LIN {X 0,Y 305.543,Z 612.418,A -85,B 0,C 180,E1 -15866.228,E2 -15866.228} C_VEL
LIN {X 0,Y 305.492,Z 612.423,A -85,B 0,C 180,E1 -15869.051,E2 -15869.051} C_VEL
LIN {X 0,Y 305.444,Z 612.427,A -85,B 0,C 180,E1 -15871.953,E2 -15871.953} C_VEL
LIN {X 0,Y 305.459,Z 612.428,A -85,B 0,C 180,E1 -15875.114,E2 -15875.114} C_VEL
LIN {X 0,Y 305.479,Z 612.428,A -85,B 0,C 180,E1 -15878.537,E2 -15878.537} C_VEL
LIN {X 0,Y 305.49,Z 612.432,A -85,B 0,C 180,E1 -15882.594,E2 -15882.594} C_VEL
LIN {X 0,Y 305.48,Z 612.432,A -85,B 0,C 180,E1 -15886.356,E2 -15886.356} C_VEL
LIN {X 0,Y 305.465,Z 612.434,A -85,B 0,C 180,E1 -15889.895,E2 -15889.895} C_VEL
LIN {X 0,Y 305.512,Z 612.46,A -85,B 0,C 180,E1 -15892.958,E2 -15892.958} C_VEL
LIN {X 0,Y 307.907,Z 621.669,A -85,B 0,C 180,E1 -15896.446,E2 -15896.446} C_VEL
LIN {X 0,Y 310.34,Z 632.372,A -85,B 0,C 180,E1 -15900.119,E2 -15900.119} C_VEL
LIN {X 0,Y 311.626,Z 639.236,A -85,B 0,C 180,E1 -15902.28,E2 -15902.28} C_VEL
LIN {X 0,Y 313.295,Z 644.798,A -85,B 0,C 180,E1 -15902.654,E2 -15902.654} C_VEL
LIN {X 0,Y 317.551,Z 667.18,A -85,B 0,C 180,E1 -15903.81,E2 -15903.81} C_VEL
LIN {X 0,Y 319.912,Z 685.577,A -85,B 0,C 180,E1 -15904.607,E2 -15904.607} C_VEL
LIN {X 0,Y 317.704,Z 749.055,A -85,B 0,C 180,E1 -15906.253,E2 -15906.253} C_VEL
LIN {X 0,Y 316.565,Z 763.423,A -85,B 0,C 180,E1 -15906.879,E2 -15906.879} C_VEL
LIN {X 0,Y 315.132,Z 776.341,A -85,B 0,C 180,E1 -15907.721,E2 -15907.721} C_VEL
LIN {X 0,Y 313.453,Z 788.638,A -85,B 0,C 180,E1 -15908.806,E2 -15908.806} C_VEL
LIN {X 0,Y 311.748,Z 799.729,A -85,B 0,C 180,E1 -15910.064,E2 -15910.064} C_VEL
LIN {X 0,Y 310.042,Z 809.772,A -85,B 0,C 180,E1 -15911.498,E2 -15911.498} C_VEL
LIN {X 0,Y 308.518,Z 818.8,A -85,B 0,C 180,E1 -15913.09,E2 -15913.09} C_VEL
LIN {X 0,Y 307.022,Z 827.902,A -85,B 0,C 180,E1 -15915.077,E2 -15915.077} C_VEL
LIN {X 0,Y 305.66,Z 835.139,A -85,B 0,C 180,E1 -15917.046,E2 -15917.046} C_VEL
LIN {X 0,Y 304.621,Z 841.793,A -85,B 0,C 180,E1 -15919.364,E2 -15919.364} C_VEL
LIN {X 0,Y 304.064,Z 846.209,A -85,B 0,C 180,E1 -15921.359,E2 -15921.359} C_VEL
LIN {X 0,Y 303.757,Z 849.545,A -85,B 0,C 180,E1 -15923.357,E2 -15923.357} C_VEL
LIN {X 0,Y 303.688,Z 851.227,A -85,B 0,C 180,E1 -15924.689,E2 -15924.689} C_VEL
LIN {X 0,Y 303.681,Z 852.481,A -85,B 0,C 180,E1 -15926.019,E2 -15926.019} C_VEL
LIN {X 0,Y 303.674,Z 853.284,A -85,B 0,C 180,E1 -15927.347,E2 -15927.347} C_VEL
LIN {X 0,Y 303.694,Z 853.688,A -85,B 0,C 180,E1 -15928.674,E2 -15928.674} C_VEL
LIN {X 0,Y 303.794,Z 853.697,A -85,B 0,C 180,E1 -15930,E2 -15930} C_VEL
LIN {X 0,Y 303.722,Z 853.275,A -85,B 0,C 180,E1 -15931.326,E2 -15931.326} C_VEL
LIN {X 0,Y 303.685,Z 852.404,A -85,B 0,C 180,E1 -15932.653,E2 -15932.653} C_VEL
LIN {X 0,Y 303.703,Z 851.122,A -85,B 0,C 180,E1 -15933.981,E2 -15933.981} C_VEL
LIN {X 0,Y 303.732,Z 848.735,A -85,B 0,C 180,E1 -15935.745,E2 -15935.745} C_VEL
LIN {X 0,Y 303.946,Z 844.524,A -85,B 0,C 180,E1 -15937.974,E2 -15937.974} C_VEL
LIN {X 0,Y 304.356,Z 839.52,A -85,B 0,C 180,E1 -15939.973,E2 -15939.973} C_VEL
LIN {X 0,Y 304.988,Z 833.193,A -85,B 0,C 180,E1 -15941.969,E2 -15941.969} C_VEL
LIN {X 0,Y 306.069,Z 825.275,A -85,B 0,C 180,E1 -15943.951,E2 -15943.951} C_VEL
LIN {X 0,Y 307.063,Z 817.151,A -85,B 0,C 180,E1 -15945.6,E2 -15945.6} C_VEL
LIN {X 0,Y 308.266,Z 807.236,A -85,B 0,C 180,E1 -15947.24,E2 -15947.24} C_VEL
LIN {X 0,Y 309.704,Z 796.205,A -85,B 0,C 180,E1 -15948.695,E2 -15948.695} C_VEL
LIN {X 0,Y 311.143,Z 783.651,A -85,B 0,C 180,E1 -15949.976,E2 -15949.976} C_VEL
LIN {X 0,Y 312.364,Z 771.376,A -85,B 0,C 180,E1 -15950.926,E2 -15950.926} C_VEL
LIN {X 0,Y 313.352,Z 758.55,A -85,B 0,C 180,E1 -15951.633,E2 -15951.633} C_VEL
LIN {X 0,Y 313.919,Z 745.321,A -85,B 0,C 180,E1 -15952.11,E2 -15952.11} C_VEL
LIN {X 0,Y 315.418,Z 683.907,A -85,B 0,C 180,E1 -15953.644,E2 -15953.644} C_VEL
LIN {X 0,Y 309.576,Z 641.497,A -85,B 0,C 180,E1 -15955.219,E2 -15955.219} C_VEL
LIN {X 0,Y 310.286,Z 636.303,A -85,B 0,C 180,E1 -15956.572,E2 -15956.572} C_VEL
LIN {X 0,Y 309.106,Z 629.471,A -85,B 0,C 180,E1 -15958.519,E2 -15958.519} C_VEL
LIN {X 0,Y 306.453,Z 617.001,A -85,B 0,C 180,E1 -15962.22,E2 -15962.22} C_VEL
LIN {X 0,Y 305.476,Z 612.433,A -85,B 0,C 180,E1 -15963.654,E2 -15963.654} C_VEL
LIN {X 0,Y 305.497,Z 612.431,A -85,B 0,C 180,E1 -15966.735,E2 -15966.735} C_VEL
LIN {X 0,Y 305.463,Z 612.438,A -85,B 0,C 180,E1 -15970.601,E2 -15970.601} C_VEL
LIN {X 0,Y 305.48,Z 612.431,A -85,B 0,C 180,E1 -15973.644,E2 -15973.644} C_VEL
LIN {X 0,Y 305.49,Z 612.429,A -85,B 0,C 180,E1 -15977.406,E2 -15977.406} C_VEL
LIN {X 0,Y 305.506,Z 612.427,A -85,B 0,C 180,E1 -15981.601,E2 -15981.601} C_VEL
LIN {X 0,Y 305.46,Z 612.438,A -85,B 0,C 180,E1 -15984.886,E2 -15984.886} C_VEL
LIN {X 0,Y 305.452,Z 612.435,A -85,B 0,C 180,E1 -15988.353,E2 -15988.353} C_VEL
LIN {X 0,Y 305.517,Z 612.429,A -85,B 0,C 180,E1 -15991.113,E2 -15991.113} C_VEL
LIN {X 0,Y 305.567,Z 612.418,A -85,B 0,C 180,E1 -15994.087,E2 -15994.087} C_VEL
LIN {X 0,Y 305.475,Z 612.431,A -85,B 0,C 180,E1 -15998.4,E2 -15998.4} C_VEL
LIN {X 0,Y 305.574,Z 612.422,A -85,B 0,C 180,E1 -16001.216,E2 -16001.216} C_VEL
LIN {X 0,Y 305.643,Z 612.414,A -85,B 0,C 180,E1 -16005.348,E2 -16005.348} C_VEL
LIN {X 0,Y 305.631,Z 612.413,A -85,B 0,C 180,E1 -16009.399,E2 -16009.399} C_VEL
LIN {X 0,Y 305.802,Z 612.389,A -85,B 0,C 180,E1 -16012.073,E2 -16012.073} C_VEL
LIN {X 0,Y 305.682,Z 612.405,A -85,B 0,C 180,E1 -16014.723,E2 -16014.723} C_VEL
LIN {X 0,Y 305.951,Z 612.371,A -85,B 0,C 180,E1 -16018.683,E2 -16018.683} C_VEL
LIN {X 0,Y 305.951,Z 612.373,A -85,B 0,C 180,E1 -16021.316,E2 -16021.316} C_VEL
LIN {X 0,Y 305.841,Z 612.385,A -85,B 0,C 180,E1 -16026.597,E2 -16026.597} C_VEL
LIN {X 0,Y 305.728,Z 612.401,A -85,B 0,C 180,E1 -16029.259,E2 -16029.259} C_VEL
LIN {X 0,Y 305.58,Z 612.416,A -85,B 0,C 180,E1 -16033.296,E2 -16033.296} C_VEL
LIN {X 0,Y 305.586,Z 612.419,A -85,B 0,C 180,E1 -16036.02,E2 -16036.02} C_VEL
LIN {X 0,Y 305.569,Z 612.421,A -85,B 0,C 180,E1 -16039.444,E2 -16039.444} C_VEL
LIN {X 0,Y 305.482,Z 612.428,A -85,B 0,C 180,E1 -16043.041,E2 -16043.041} C_VEL
LIN {X 0,Y 305.54,Z 612.423,A -85,B 0,C 180,E1 -16046.227,E2 -16046.227} C_VEL
LIN {X 0,Y 305.488,Z 612.428,A -85,B 0,C 180,E1 -16049.05,E2 -16049.05} C_VEL
LIN {X 0,Y 305.441,Z 612.439,A -85,B 0,C 180,E1 -16051.952,E2 -16051.952} C_VEL
LIN {X 0,Y 305.455,Z 612.432,A -85,B 0,C 180,E1 -16055.113,E2 -16055.113} C_VEL
LIN {X 0,Y 305.486,Z 612.429,A -85,B 0,C 180,E1 -16058.539,E2 -16058.539} C_VEL
LIN {X 0,Y 305.504,Z 612.429,A -85,B 0,C 180,E1 -16062.597,E2 -16062.597} C_VEL
LIN {X 0,Y 305.481,Z 612.434,A -85,B 0,C 180,E1 -16066.356,E2 -16066.356} C_VEL
LIN {X 0,Y 305.459,Z 612.431,A -85,B 0,C 180,E1 -16069.894,E2 -16069.894} C_VEL
LIN {X 0,Y 305.494,Z 612.428,A -85,B 0,C 180,E1 -16073.627,E2 -16073.627} C_VEL
LIN {X 0,Y 305.46,Z 612.438,A -85,B 0,C 180,E1 -16076.484,E2 -16076.484} C_VEL
LIN {X 0,Y 305.452,Z 612.431,A -85,B 0,C 180,E1 -16079.591,E2 -16079.591} C_VEL
LIN {X 0,Y 305.51,Z 612.432,A -85,B 0,C 180,E1 -16082.608,E2 -16082.608} C_VEL
LIN {X 0,Y 305.503,Z 612.427,A -85,B 0,C 180,E1 -16085.539,E2 -16085.539} C_VEL
LIN {X 0,Y 305.516,Z 612.425,A -85,B 0,C 180,E1 -16089.815,E2 -16089.815} C_VEL
LIN {X 0,Y 305.571,Z 612.423,A -85,B 0,C 180,E1 -16092.603,E2 -16092.603} C_VEL
LIN {X 0,Y 305.645,Z 612.41,A -85,B 0,C 180,E1 -16095.349,E2 -16095.349} C_VEL
LIN {X 0,Y 305.635,Z 612.411,A -85,B 0,C 180,E1 -16099.4,E2 -16099.4} C_VEL
LIN {X 0,Y 305.805,Z 612.389,A -85,B 0,C 180,E1 -16102.074,E2 -16102.074} C_VEL
LIN {X 0,Y 305.685,Z 612.407,A -85,B 0,C 180,E1 -16104.724,E2 -16104.724} C_VEL
LIN {X 0,Y 305.955,Z 612.373,A -85,B 0,C 180,E1 -16108.684,E2 -16108.684} C_VEL
LIN {X 0,Y 305.955,Z 612.374,A -85,B 0,C 180,E1 -16111.316,E2 -16111.316} C_VEL
LIN {X 0,Y 305.684,Z 612.409,A -85,B 0,C 180,E1 -16115.276,E2 -16115.276} C_VEL
LIN {X 0,Y 305.793,Z 612.392,A -85,B 0,C 180,E1 -16117.926,E2 -16117.926} C_VEL
LIN {X 0,Y 305.6,Z 612.416,A -85,B 0,C 180,E1 -16121.945,E2 -16121.945} C_VEL
LIN {X 0,Y 305.634,Z 612.415,A -85,B 0,C 180,E1 -16125.035,E2 -16125.035} C_VEL
LIN {X 0,Y 305.633,Z 612.47,A -85,B 0,C 180,E1 -16129.167,E2 -16129.167} C_VEL
LIN {X 0,Y 305.85,Z 613.833,A -85,B 0,C 180,E1 -16129.639,E2 -16129.639} C_VEL
LIN {X 0,Y 316.129,Z 642.397,A -85,B 0,C 180,E1 -16131.156,E2 -16131.156} C_VEL
LIN {X 0,Y 315.453,Z 671.633,A -85,B 0,C 180,E1 -16131.889,E2 -16131.889} C_VEL
LIN {X 0,Y 313.978,Z 721.477,A -85,B 0,C 180,E1 -16133.152,E2 -16133.152} C_VEL
LIN {X 0,Y 313.316,Z 735.297,A -85,B 0,C 180,E1 -16133.778,E2 -16133.778} C_VEL
LIN {X 0,Y 312.468,Z 747.528,A -85,B 0,C 180,E1 -16134.588,E2 -16134.588} C_VEL
LIN {X 0,Y 311.433,Z 758.765,A -85,B 0,C 180,E1 -16135.576,E2 -16135.576} C_VEL
LIN {X 0,Y 310.359,Z 769.3,A -85,B 0,C 180,E1 -16136.751,E2 -16136.751} C_VEL
LIN {X 0,Y 309.152,Z 778.865,A -85,B 0,C 180,E1 -16138.06,E2 -16138.06} C_VEL
LIN {X 0,Y 308.068,Z 788.02,A -85,B 0,C 180,E1 -16139.597,E2 -16139.597} C_VEL
LIN {X 0,Y 306.895,Z 796.747,A -85,B 0,C 180,E1 -16141.397,E2 -16141.397} C_VEL
LIN {X 0,Y 305.795,Z 804.771,A -85,B 0,C 180,E1 -16143.475,E2 -16143.475} C_VEL
LIN {X 0,Y 304.953,Z 811.468,A -85,B 0,C 180,E1 -16145.676,E2 -16145.676} C_VEL
LIN {X 0,Y 304.418,Z 815.911,A -85,B 0,C 180,E1 -16147.554,E2 -16147.554} C_VEL
LIN {X 0,Y 304.021,Z 819.316,A -85,B 0,C 180,E1 -16149.417,E2 -16149.417} C_VEL
LIN {X 0,Y 303.747,Z 821.79,A -85,B 0,C 180,E1 -16151.255,E2 -16151.255} C_VEL
LIN {X 0,Y 303.507,Z 823.992,A -85,B 0,C 180,E1 -16154,E2 -16154} C_VEL
LIN {X 0,Y 303.51,Z 824.497,A -85,B 0,C 180,E1 -16156,E2 -16156} C_VEL
LIN {X 0,Y 303.647,Z 824.132,A -85,B 0,C 180,E1 -16157.84,E2 -16157.84} C_VEL
LIN {X 0,Y 303.992,Z 822.94,A -85,B 0,C 180,E1 -16159.721,E2 -16159.721} C_VEL
LIN {X 0,Y 304.443,Z 820.788,A -85,B 0,C 180,E1 -16161.708,E2 -16161.708} C_VEL
LIN {X 0,Y 305.069,Z 817.577,A -85,B 0,C 180,E1 -16163.735,E2 -16163.735} C_VEL
LIN {X 0,Y 306.122,Z 812.196,A -85,B 0,C 180,E1 -16166.19,E2 -16166.19} C_VEL
LIN {X 0,Y 307.281,Z 806.133,A -85,B 0,C 180,E1 -16168.262,E2 -16168.262} C_VEL
LIN {X 0,Y 308.82,Z 798.31,A -85,B 0,C 180,E1 -16170.361,E2 -16170.361} C_VEL
LIN {X 0,Y 310.445,Z 789.859,A -85,B 0,C 180,E1 -16172.164,E2 -16172.164} C_VEL
LIN {X 0,Y 311.242,Z 785.111,A -85,B 0,C 180,E1 -16173.023,E2 -16173.023} C_VEL
LIN {X 0,Y 311.3,Z 780.871,A -85,B 0,C 180,E1 -16173.773,E2 -16173.773} C_VEL
LIN {X 0,Y 309.142,Z 770.889,A -85,B 0,C 180,E1 -16175.515,E2 -16175.515} C_VEL
LIN {X 0,Y 308.347,Z 764.725,A -85,B 0,C 180,E1 -16176.411,E2 -16176.411} C_VEL
LIN {X 0,Y 308.54,Z 761.356,A -85,B 0,C 180,E1 -16176.796,E2 -16176.796} C_VEL
LIN {X 0,Y 310.052,Z 749.256,A -85,B 0,C 180,E1 -16177.895,E2 -16177.895} C_VEL
LIN {X 0,Y 311.225,Z 735.781,A -85,B 0,C 180,E1 -16178.795,E2 -16178.795} C_VEL
LIN {X 0,Y 312.046,Z 722.907,A -85,B 0,C 180,E1 -16179.377,E2 -16179.377} C_VEL
LIN {X 0,Y 314.81,Z 649.184,A -85,B 0,C 180,E1 -16181.33,E2 -16181.33} C_VEL
LIN {X 0,Y 308.378,Z 634.264,A -85,B 0,C 180,E1 -16182.569,E2 -16182.569} C_VEL
LIN {X 0,Y 301.448,Z 620.861,A -85,B 0,C 180,E1 -16183.918,E2 -16183.918} C_VEL
LIN {X 0,Y 299.513,Z 617.125,A -85,B 0,C 180,E1 -16184.346,E2 -16184.346} C_VEL
LIN {X 0,Y 298.551,Z 613.297,A -85,B 0,C 180,E1 -16186.212,E2 -16186.212} C_VEL
LIN {X 0,Y 298.753,Z 613.274,A -85,B 0,C 180,E1 -16191.115,E2 -16191.115} C_VEL
LIN {X 0,Y 298.792,Z 613.269,A -85,B 0,C 180,E1 -16193.247,E2 -16193.247} C_VEL
LIN {X 0,Y 298.85,Z 613.26,A -85,B 0,C 180,E1 -16197.305,E2 -16197.305} C_VEL
LIN {X 0,Y 299.019,Z 613.238,A -85,B 0,C 180,E1 -16200.001,E2 -16200.001} C_VEL
LIN {X 0,Y 298.842,Z 613.262,A -85,B 0,C 180,E1 -16202.697,E2 -16202.697} C_VEL
LIN {X 0,Y 298.793,Z 613.262,A -85,B 0,C 180,E1 -16206.755,E2 -16206.755} C_VEL
LIN {X 0,Y 298.675,Z 613.275,A -85,B 0,C 180,E1 -16209.481,E2 -16209.481} C_VEL
LIN {X 0,Y 298.547,Z 613.294,A -85,B 0,C 180,E1 -16213.616,E2 -16213.616} C_VEL
LIN {X 0,Y 298.543,Z 613.29,A -85,B 0,C 180,E1 -16216.41,E2 -16216.41} C_VEL
LIN {X 0,Y 298.506,Z 613.297,A -85,B 0,C 180,E1 -16219.656,E2 -16219.656} C_VEL
LIN {X 0,Y 298.453,Z 613.307,A -85,B 0,C 180,E1 -16223.599,E2 -16223.599} C_VEL
LIN {X 0,Y 298.485,Z 613.298,A -85,B 0,C 180,E1 -16226.575,E2 -16226.575} C_VEL
LIN {X 0,Y 298.418,Z 613.306,A -85,B 0,C 180,E1 -16229.642,E2 -16229.642} C_VEL
LIN {X 0,Y 298.394,Z 613.308,A -85,B 0,C 180,E1 -16232.801,E2 -16232.801} C_VEL
LIN {X 0,Y 298.462,Z 613.306,A -85,B 0,C 180,E1 -16236.814,E2 -16236.814} C_VEL
LIN {X 0,Y 298.416,Z 613.308,A -85,B 0,C 180,E1 -16241.096,E2 -16241.096} C_VEL
LIN {X 0,Y 298.416,Z 613.315,A -85,B 0,C 180,E1 -16245.048,E2 -16245.048} C_VEL
LIN {X 0,Y 298.419,Z 613.314,A -85,B 0,C 180,E1 -16248.746,E2 -16248.746} C_VEL
LIN {X 0,Y 298.467,Z 613.386,A -85,B 0,C 180,E1 -16252.091,E2 -16252.091} C_VEL
LIN {X 0,Y 301.004,Z 623.033,A -85,B 0,C 180,E1 -16255.92,E2 -16255.92} C_VEL
LIN {X 0,Y 303.174,Z 632.6,A -85,B 0,C 180,E1 -16259.338,E2 -16259.338} C_VEL
LIN {X 0,Y 304.453,Z 638.904,A -85,B 0,C 180,E1 -16261.378,E2 -16261.378} C_VEL
LIN {X 0,Y 307.133,Z 645.608,A -85,B 0,C 180,E1 -16261.934,E2 -16261.934} C_VEL
LIN {X 0,Y 310.973,Z 665.162,A -85,B 0,C 180,E1 -16263.018,E2 -16263.018} C_VEL
LIN {X 0,Y 313.303,Z 682.326,A -85,B 0,C 180,E1 -16263.804,E2 -16263.804} C_VEL
LIN {X 0,Y 313.776,Z 686.682,A -85,B 0,C 180,E1 -16263.987,E2 -16263.987} C_VEL
LIN {X 0,Y 311.45,Z 748.992,A -85,B 0,C 180,E1 -16265.642,E2 -16265.642} C_VEL
LIN {X 0,Y 310.314,Z 762.71,A -85,B 0,C 180,E1 -16266.253,E2 -16266.253} C_VEL
LIN {X 0,Y 308.881,Z 775.201,A -85,B 0,C 180,E1 -16267.068,E2 -16267.068} C_VEL
LIN {X 0,Y 307.143,Z 787.602,A -85,B 0,C 180,E1 -16268.172,E2 -16268.172} C_VEL
LIN {X 0,Y 305.355,Z 798.807,A -85,B 0,C 180,E1 -16269.453,E2 -16269.453} C_VEL
LIN {X 0,Y 303.516,Z 808.983,A -85,B 0,C 180,E1 -16270.91,E2 -16270.91} C_VEL
LIN {X 0,Y 301.801,Z 818.419,A -85,B 0,C 180,E1 -16272.598,E2 -16272.598} C_VEL
LIN {X 0,Y 300.335,Z 826.557,A -85,B 0,C 180,E1 -16274.389,E2 -16274.389} C_VEL
LIN {X 0,Y 298.948,Z 833.99,A -85,B 0,C 180,E1 -16276.403,E2 -16276.403} C_VEL
LIN {X 0,Y 297.852,Z 839.972,A -85,B 0,C 180,E1 -16278.43,E2 -16278.43} C_VEL
LIN {X 0,Y 297.198,Z 844.71,A -85,B 0,C 180,E1 -16280.472,E2 -16280.472} C_VEL
LIN {X 0,Y 296.789,Z 848.348,A -85,B 0,C 180,E1 -16282.517,E2 -16282.517} C_VEL
LIN {X 0,Y 296.603,Z 850.97,A -85,B 0,C 180,E1 -16284.561,E2 -16284.561} C_VEL
LIN {X 0,Y 296.596,Z 852.183,A -85,B 0,C 180,E1 -16285.924,E2 -16285.924} C_VEL
LIN {X 0,Y 296.597,Z 852.965,A -85,B 0,C 180,E1 -16287.284,E2 -16287.284} C_VEL
LIN {X 0,Y 296.607,Z 853.349,A -85,B 0,C 180,E1 -16288.642,E2 -16288.642} C_VEL
LIN {X 0,Y 296.702,Z 853.337,A -85,B 0,C 180,E1 -16290,E2 -16290} C_VEL
LIN {X 0,Y 296.633,Z 852.871,A -85,B 0,C 180,E1 -16291.358,E2 -16291.358} C_VEL
LIN {X 0,Y 296.608,Z 851.976,A -85,B 0,C 180,E1 -16292.716,E2 -16292.716} C_VEL
LIN {X 0,Y 296.616,Z 850.67,A -85,B 0,C 180,E1 -16294.076,E2 -16294.076} C_VEL
LIN {X 0,Y 296.631,Z 848.565,A -85,B 0,C 180,E1 -16295.672,E2 -16295.672} C_VEL
LIN {X 0,Y 296.885,Z 843.967,A -85,B 0,C 180,E1 -16298.165,E2 -16298.165} C_VEL
LIN {X 0,Y 297.341,Z 838.904,A -85,B 0,C 180,E1 -16300.211,E2 -16300.211} C_VEL
LIN {X 0,Y 298.007,Z 832.506,A -85,B 0,C 180,E1 -16302.254,E2 -16302.254} C_VEL
LIN {X 0,Y 299.085,Z 824.47,A -85,B 0,C 180,E1 -16304.284,E2 -16304.284} C_VEL
LIN {X 0,Y 300.065,Z 816.867,A -85,B 0,C 180,E1 -16305.856,E2 -16305.856} C_VEL
LIN {X 0,Y 301.422,Z 806.228,A -85,B 0,C 180,E1 -16307.644,E2 -16307.644} C_VEL
LIN {X 0,Y 302.906,Z 794.975,A -85,B 0,C 180,E1 -16309.13,E2 -16309.13} C_VEL
LIN {X 0,Y 304.245,Z 783.988,A -85,B 0,C 180,E1 -16310.273,E2 -16310.273} C_VEL
LIN {X 0,Y 305.496,Z 771.915,A -85,B 0,C 180,E1 -16311.243,E2 -16311.243} C_VEL
LIN {X 0,Y 306.506,Z 759.574,A -85,B 0,C 180,E1 -16311.964,E2 -16311.964} C_VEL
LIN {X 0,Y 307.153,Z 745.761,A -85,B 0,C 180,E1 -16312.491,E2 -16312.491} C_VEL
LIN {X 0,Y 308.682,Z 684.406,A -85,B 0,C 180,E1 -16314.064,E2 -16314.064} C_VEL
LIN {X 0,Y 302.771,Z 641.232,A -85,B 0,C 180,E1 -16315.711,E2 -16315.711} C_VEL
LIN {X 0,Y 303.276,Z 636.934,A -85,B 0,C 180,E1 -16316.864,E2 -16316.864} C_VEL
LIN {X 0,Y 301.412,Z 627.069,A -85,B 0,C 180,E1 -16319.764,E2 -16319.764} C_VEL
LIN {X 0,Y 298.431,Z 613.311,A -85,B 0,C 180,E1 -16324.058,E2 -16324.058} C_VEL
LIN {X 0,Y 298.439,Z 613.307,A -85,B 0,C 180,E1 -16327.753,E2 -16327.753} C_VEL
LIN {X 0,Y 298.419,Z 613.311,A -85,B 0,C 180,E1 -16331.254,E2 -16331.254} C_VEL
LIN {X 0,Y 298.415,Z 613.313,A -85,B 0,C 180,E1 -16335.046,E2 -16335.046} C_VEL
LIN {X 0,Y 298.416,Z 613.314,A -85,B 0,C 180,E1 -16338.904,E2 -16338.904} C_VEL
LIN {X 0,Y 298.464,Z 613.307,A -85,B 0,C 180,E1 -16343.186,E2 -16343.186} C_VEL
LIN {X 0,Y 298.394,Z 613.315,A -85,B 0,C 180,E1 -16347.199,E2 -16347.199} C_VEL
LIN {X 0,Y 298.429,Z 613.311,A -85,B 0,C 180,E1 -16350.613,E2 -16350.613} C_VEL
LIN {X 0,Y 298.48,Z 613.302,A -85,B 0,C 180,E1 -16353.473,E2 -16353.473} C_VEL
LIN {X 0,Y 298.426,Z 613.311,A -85,B 0,C 180,E1 -16356.699,E2 -16356.699} C_VEL
LIN {X 0,Y 298.52,Z 613.299,A -85,B 0,C 180,E1 -16360.755,E2 -16360.755} C_VEL
LIN {X 0,Y 298.587,Z 613.292,A -85,B 0,C 180,E1 -16364.994,E2 -16364.994} C_VEL
LIN {X 0,Y 298.587,Z 613.293,A -85,B 0,C 180,E1 -16369.146,E2 -16369.146} C_VEL
LIN {X 0,Y 298.748,Z 613.268,A -85,B 0,C 180,E1 -16371.885,E2 -16371.885} C_VEL
LIN {X 0,Y 298.653,Z 613.281,A -85,B 0,C 180,E1 -16374.598,E2 -16374.598} C_VEL
LIN {X 0,Y 298.918,Z 613.247,A -85,B 0,C 180,E1 -16378.652,E2 -16378.652} C_VEL
LIN {X 0,Y 298.918,Z 613.249,A -85,B 0,C 180,E1 -16381.347,E2 -16381.347} C_VEL
LIN {X 0,Y 298.787,Z 613.264,A -85,B 0,C 180,E1 -16386.753,E2 -16386.753} C_VEL
LIN {X 0,Y 298.673,Z 613.282,A -85,B 0,C 180,E1 -16389.48,E2 -16389.48} C_VEL
LIN {X 0,Y 298.544,Z 613.294,A -85,B 0,C 180,E1 -16393.615,E2 -16393.615} C_VEL
LIN {X 0,Y 298.541,Z 613.294,A -85,B 0,C 180,E1 -16396.408,E2 -16396.408} C_VEL
LIN {X 0,Y 298.504,Z 613.303,A -85,B 0,C 180,E1 -16399.654,E2 -16399.654} C_VEL
LIN {X 0,Y 298.45,Z 613.307,A -85,B 0,C 180,E1 -16403.598,E2 -16403.598} C_VEL
LIN {X 0,Y 298.482,Z 613.299,A -85,B 0,C 180,E1 -16406.574,E2 -16406.574} C_VEL
LIN {X 0,Y 298.414,Z 613.311,A -85,B 0,C 180,E1 -16409.641,E2 -16409.641} C_VEL
LIN {X 0,Y 298.39,Z 613.313,A -85,B 0,C 180,E1 -16412.8,E2 -16412.8} C_VEL
LIN {X 0,Y 298.463,Z 613.301,A -85,B 0,C 180,E1 -16416.814,E2 -16416.814} C_VEL
LIN {X 0,Y 298.446,Z 613.305,A -85,B 0,C 180,E1 -16421.25,E2 -16421.25} C_VEL
LIN {X 0,Y 298.411,Z 613.31,A -85,B 0,C 180,E1 -16425.047,E2 -16425.047} C_VEL
LIN {X 0,Y 298.414,Z 613.309,A -85,B 0,C 180,E1 -16428.745,E2 -16428.745} C_VEL
LIN {X 0,Y 298.433,Z 613.31,A -85,B 0,C 180,E1 -16432.246,E2 -16432.246} C_VEL
LIN {X 0,Y 298.403,Z 613.312,A -85,B 0,C 180,E1 -16435.581,E2 -16435.581} C_VEL
LIN {X 0,Y 298.386,Z 613.314,A -85,B 0,C 180,E1 -16438.791,E2 -16438.791} C_VEL
LIN {X 0,Y 298.452,Z 613.305,A -85,B 0,C 180,E1 -16441.904,E2 -16441.904} C_VEL
LIN {X 0,Y 298.479,Z 613.304,A -85,B 0,C 180,E1 -16444.924,E2 -16444.924} C_VEL
LIN {X 0,Y 298.446,Z 613.307,A -85,B 0,C 180,E1 -16449.316,E2 -16449.316} C_VEL
LIN {X 0,Y 298.534,Z 613.296,A -85,B 0,C 180,E1 -16452.18,E2 -16452.18} C_VEL
LIN {X 0,Y 298.59,Z 613.291,A -85,B 0,C 180,E1 -16454.995,E2 -16454.995} C_VEL
LIN {X 0,Y 298.59,Z 613.291,A -85,B 0,C 180,E1 -16459.147,E2 -16459.147} C_VEL
LIN {X 0,Y 298.751,Z 613.267,A -85,B 0,C 180,E1 -16461.886,E2 -16461.886} C_VEL
LIN {X 0,Y 298.655,Z 613.282,A -85,B 0,C 180,E1 -16464.599,E2 -16464.599} C_VEL
LIN {X 0,Y 298.921,Z 613.248,A -85,B 0,C 180,E1 -16468.653,E2 -16468.653} C_VEL
LIN {X 0,Y 298.921,Z 613.25,A -85,B 0,C 180,E1 -16471.347,E2 -16471.347} C_VEL
LIN {X 0,Y 298.784,Z 613.266,A -85,B 0,C 180,E1 -16476.754,E2 -16476.754} C_VEL
LIN {X 0,Y 298.632,Z 613.287,A -85,B 0,C 180,E1 -16479.482,E2 -16479.482} C_VEL
LIN {X 0,Y 298.549,Z 613.298,A -85,B 0,C 180,E1 -16483.615,E2 -16483.615} C_VEL
LIN {X 0,Y 298.546,Z 613.295,A -85,B 0,C 180,E1 -16486.408,E2 -16486.408} C_VEL
LIN {X 0,Y 298.577,Z 613.417,A -85,B 0,C 180,E1 -16488.839,E2 -16488.839} C_VEL
LIN {X 0,Y 298.714,Z 614.142,A -85,B 0,C 180,E1 -16489.097,E2 -16489.097} C_VEL
LIN {X 0,Y 309.479,Z 643.855,A -85,B 0,C 180,E1 -16490.739,E2 -16490.739} C_VEL
LIN {X 0,Y 307.27,Z 721.207,A -85,B 0,C 180,E1 -16492.73,E2 -16492.73} C_VEL
LIN {X 0,Y 306.588,Z 734.937,A -85,B 0,C 180,E1 -16493.354,E2 -16493.354} C_VEL
LIN {X 0,Y 305.698,Z 747.493,A -85,B 0,C 180,E1 -16494.189,E2 -16494.189} C_VEL
LIN {X 0,Y 304.559,Z 759.516,A -85,B 0,C 180,E1 -16495.271,E2 -16495.271} C_VEL
LIN {X 0,Y 303.43,Z 770.04,A -85,B 0,C 180,E1 -16496.478,E2 -16496.478} C_VEL
LIN {X 0,Y 302.143,Z 779.991,A -85,B 0,C 180,E1 -16497.885,E2 -16497.885} C_VEL
LIN {X 0,Y 301.104,Z 788.435,A -85,B 0,C 180,E1 -16499.35,E2 -16499.35} C_VEL
LIN {X 0,Y 299.82,Z 797.74,A -85,B 0,C 180,E1 -16501.336,E2 -16501.336} C_VEL
LIN {X 0,Y 298.847,Z 804.585,A -85,B 0,C 180,E1 -16503.145,E2 -16503.145} C_VEL
LIN {X 0,Y 298.005,Z 811.107,A -85,B 0,C 180,E1 -16505.294,E2 -16505.294} C_VEL
LIN {X 0,Y 297.429,Z 815.684,A -85,B 0,C 180,E1 -16507.209,E2 -16507.209} C_VEL
LIN {X 0,Y 297.076,Z 818.523,A -85,B 0,C 180,E1 -16508.677,E2 -16508.677} C_VEL
LIN {X 0,Y 296.71,Z 821.532,A -85,B 0,C 180,E1 -16510.716,E2 -16510.716} C_VEL
LIN {X 0,Y 296.425,Z 823.996,A -85,B 0,C 180,E1 -16513.436,E2 -16513.436} C_VEL
LIN {X 0,Y 296.381,Z 824.753,A -85,B 0,C 180,E1 -16515.346,E2 -16515.346} C_VEL
LIN {X 0,Y 296.489,Z 824.712,A -85,B 0,C 180,E1 -16517.291,E2 -16517.291} C_VEL
LIN {X 0,Y 296.814,Z 823.82,A -85,B 0,C 180,E1 -16519.26,E2 -16519.26} C_VEL
LIN {X 0,Y 297.264,Z 821.997,A -85,B 0,C 180,E1 -16521.277,E2 -16521.277} C_VEL
LIN {X 0,Y 298.04,Z 818.231,A -85,B 0,C 180,E1 -16523.878,E2 -16523.878} C_VEL
LIN {X 0,Y 298.995,Z 813.721,A -85,B 0,C 180,E1 -16526.066,E2 -16526.066} C_VEL
LIN {X 0,Y 300.229,Z 807.64,A -85,B 0,C 180,E1 -16528.314,E2 -16528.314} C_VEL
LIN {X 0,Y 301.825,Z 799.991,A -85,B 0,C 180,E1 -16530.485,E2 -16530.485} C_VEL
LIN {X 0,Y 303.604,Z 791.35,A -85,B 0,C 180,E1 -16532.422,E2 -16532.422} C_VEL
LIN {X 0,Y 305.235,Z 782.329,A -85,B 0,C 180,E1 -16534.058,E2 -16534.058} C_VEL
LIN {X 0,Y 307.102,Z 771.099,A -85,B 0,C 180,E1 -16535.675,E2 -16535.675} C_VEL
LIN {X 0,Y 308.54,Z 761.356,A -85,B 0,C 180,E1 -16536.796,E2 -16536.796} C_VEL
LIN {X 0,Y 308.675,Z 756.268,A -85,B 0,C 180,E1 -16537.352,E2 -16537.352} C_VEL
LIN {X 0,Y 307.227,Z 747.915,A -85,B 0,C 180,E1 -16538.302,E2 -16538.302} C_VEL
LIN {X 0,Y 305.534,Z 739.304,A -85,B 0,C 180,E1 -16539.165,E2 -16539.165} C_VEL
LIN {X 0,Y 305.17,Z 733.808,A -85,B 0,C 180,E1 -16539.565,E2 -16539.565} C_VEL
LIN {X 0,Y 306.01,Z 720.628,A -85,B 0,C 180,E1 -16540.108,E2 -16540.108} C_VEL
LIN {X 0,Y 308.78,Z 651.206,A -85,B 0,C 180,E1 -16541.978,E2 -16541.978} C_VEL
LIN {X 0,Y 302.791,Z 637.387,A -85,B 0,C 180,E1 -16543.178,E2 -16543.178} C_VEL
LIN {X 0,Y 296.387,Z 624.948,A -85,B 0,C 180,E1 -16544.488,E2 -16544.488} C_VEL
LIN {X 0,Y 292.396,Z 617.603,A -85,B 0,C 180,E1 -16545.383,E2 -16545.383} C_VEL
LIN {X 0,Y 291.487,Z 614.177,A -85,B 0,C 180,E1 -16547.114,E2 -16547.114} C_VEL
LIN {X 0,Y 291.702,Z 614.152,A -85,B 0,C 180,E1 -16551.689,E2 -16551.689} C_VEL
LIN {X 0,Y 291.629,Z 614.157,A -85,B 0,C 180,E1 -16554.469,E2 -16554.469} C_VEL
LIN {X 0,Y 291.888,Z 614.124,A -85,B 0,C 180,E1 -16558.621,E2 -16558.621} C_VEL
LIN {X 0,Y 291.887,Z 614.123,A -85,B 0,C 180,E1 -16561.38,E2 -16561.38} C_VEL
LIN {X 0,Y 291.741,Z 614.14,A -85,B 0,C 180,E1 -16566.919,E2 -16566.919} C_VEL
LIN {X 0,Y 291.624,Z 614.153,A -85,B 0,C 180,E1 -16569.713,E2 -16569.713} C_VEL
LIN {X 0,Y 291.517,Z 614.172,A -85,B 0,C 180,E1 -16573.951,E2 -16573.951} C_VEL
LIN {X 0,Y 291.481,Z 614.172,A -85,B 0,C 180,E1 -16576.819,E2 -16576.819} C_VEL
LIN {X 0,Y 291.446,Z 614.178,A -85,B 0,C 180,E1 -16579.876,E2 -16579.876} C_VEL
LIN {X 0,Y 291.396,Z 614.186,A -85,B 0,C 180,E1 -16584.206,E2 -16584.206} C_VEL
LIN {X 0,Y 291.419,Z 614.184,A -85,B 0,C 180,E1 -16587.273,E2 -16587.273} C_VEL
LIN {X 0,Y 291.336,Z 614.191,A -85,B 0,C 180,E1 -16590.438,E2 -16590.438} C_VEL
LIN {X 0,Y 291.342,Z 614.191,A -85,B 0,C 180,E1 -16593.699,E2 -16593.699} C_VEL
LIN {X 0,Y 291.395,Z 614.183,A -85,B 0,C 180,E1 -16597.261,E2 -16597.261} C_VEL
LIN {X 0,Y 291.374,Z 614.185,A -85,B 0,C 180,E1 -16600.636,E2 -16600.636} C_VEL
LIN {X 0,Y 291.341,Z 614.195,A -85,B 0,C 180,E1 -16604.393,E2 -16604.393} C_VEL
LIN {X 0,Y 291.356,Z 614.192,A -85,B 0,C 180,E1 -16608.399,E2 -16608.399} C_VEL
LIN {X 0,Y 291.411,Z 614.359,A -85,B 0,C 180,E1 -16611.169,E2 -16611.169} C_VEL
LIN {X 0,Y 293.577,Z 622.215,A -85,B 0,C 180,E1 -16614.483,E2 -16614.483} C_VEL
LIN {X 0,Y 295.546,Z 630.518,A -85,B 0,C 180,E1 -16617.654,E2 -16617.654} C_VEL
LIN {X 0,Y 297.187,Z 638.246,A -85,B 0,C 180,E1 -16620.376,E2 -16620.376} C_VEL
LIN {X 0,Y 301.483,Z 648.322,A -85,B 0,C 180,E1 -16621.302,E2 -16621.302} C_VEL
LIN {X 0,Y 305.073,Z 666.958,A -85,B 0,C 180,E1 -16622.366,E2 -16622.366} C_VEL
LIN {X 0,Y 307.223,Z 683.292,A -85,B 0,C 180,E1 -16623.147,E2 -16623.147} C_VEL
LIN {X 0,Y 307.616,Z 688.615,A -85,B 0,C 180,E1 -16623.361,E2 -16623.361} C_VEL
LIN {X 0,Y 305.25,Z 748.282,A -85,B 0,C 180,E1 -16624.973,E2 -16624.973} C_VEL
LIN {X 0,Y 304.13,Z 762.139,A -85,B 0,C 180,E1 -16625.603,E2 -16625.603} C_VEL
LIN {X 0,Y 302.683,Z 774.186,A -85,B 0,C 180,E1 -16626.389,E2 -16626.389} C_VEL
LIN {X 0,Y 300.841,Z 786.731,A -85,B 0,C 180,E1 -16627.51,E2 -16627.51} C_VEL
LIN {X 0,Y 298.995,Z 797.996,A -85,B 0,C 180,E1 -16628.815,E2 -16628.815} C_VEL
LIN {X 0,Y 297.011,Z 808.245,A -85,B 0,C 180,E1 -16630.295,E2 -16630.295} C_VEL
LIN {X 0,Y 295.236,Z 817.506,A -85,B 0,C 180,E1 -16631.974,E2 -16631.974} C_VEL
LIN {X 0,Y 293.462,Z 826.597,A -85,B 0,C 180,E1 -16634.014,E2 -16634.014} C_VEL
LIN {X 0,Y 292.024,Z 833.962,A -85,B 0,C 180,E1 -16636.075,E2 -16636.075} C_VEL
LIN {X 0,Y 290.871,Z 839.869,A -85,B 0,C 180,E1 -16638.149,E2 -16638.149} C_VEL
LIN {X 0,Y 290.155,Z 844.549,A -85,B 0,C 180,E1 -16640.239,E2 -16640.239} C_VEL
LIN {X 0,Y 289.717,Z 848.138,A -85,B 0,C 180,E1 -16642.333,E2 -16642.333} C_VEL
LIN {X 0,Y 289.519,Z 850.717,A -85,B 0,C 180,E1 -16644.428,E2 -16644.428} C_VEL
LIN {X 0,Y 289.494,Z 851.886,A -85,B 0,C 180,E1 -16645.824,E2 -16645.824} C_VEL
LIN {X 0,Y 289.521,Z 852.648,A -85,B 0,C 180,E1 -16647.217,E2 -16647.217} C_VEL
LIN {X 0,Y 289.522,Z 853.011,A -85,B 0,C 180,E1 -16648.609,E2 -16648.609} C_VEL
LIN {X 0,Y 289.61,Z 852.971,A -85,B 0,C 180,E1 -16650,E2 -16650} C_VEL
LIN {X 0,Y 289.547,Z 852.466,A -85,B 0,C 180,E1 -16651.391,E2 -16651.391} C_VEL
LIN {X 0,Y 289.533,Z 851.55,A -85,B 0,C 180,E1 -16652.783,E2 -16652.783} C_VEL
LIN {X 0,Y 289.532,Z 850.219,A -85,B 0,C 180,E1 -16654.176,E2 -16654.176} C_VEL
LIN {X 0,Y 289.579,Z 847.354,A -85,B 0,C 180,E1 -16656.269,E2 -16656.269} C_VEL
LIN {X 0,Y 289.842,Z 843.41,A -85,B 0,C 180,E1 -16658.365,E2 -16658.365} C_VEL
LIN {X 0,Y 290.407,Z 837.294,A -85,B 0,C 180,E1 -16660.81,E2 -16660.81} C_VEL
LIN {X 0,Y 291.242,Z 830.55,A -85,B 0,C 180,E1 -16662.897,E2 -16662.897} C_VEL
LIN {X 0,Y 292.387,Z 822.157,A -85,B 0,C 180,E1 -16664.974,E2 -16664.974} C_VEL
LIN {X 0,Y 293.472,Z 813.517,A -85,B 0,C 180,E1 -16666.7,E2 -16666.7} C_VEL
LIN {X 0,Y 294.892,Z 802.847,A -85,B 0,C 180,E1 -16668.407,E2 -16668.407} C_VEL
LIN {X 0,Y 296.345,Z 792.319,A -85,B 0,C 180,E1 -16669.751,E2 -16669.751} C_VEL
LIN {X 0,Y 297.71,Z 780.738,A -85,B 0,C 180,E1 -16670.919,E2 -16670.919} C_VEL
LIN {X 0,Y 299.017,Z 767.546,A -85,B 0,C 180,E1 -16671.908,E2 -16671.908} C_VEL
LIN {X 0,Y 300.051,Z 754.382,A -85,B 0,C 180,E1 -16672.598,E2 -16672.598} C_VEL
LIN {X 0,Y 300.643,Z 738.519,A -85,B 0,C 180,E1 -16673.096,E2 -16673.096} C_VEL
LIN {X 0,Y 301.991,Z 685.153,A -85,B 0,C 180,E1 -16674.497,E2 -16674.497} C_VEL
LIN {X 0,Y 295.947,Z 640.938,A -85,B 0,C 180,E1 -16676.22,E2 -16676.22} C_VEL
LIN {X 0,Y 296.221,Z 637.499,A -85,B 0,C 180,E1 -16677.175,E2 -16677.175} C_VEL
LIN {X 0,Y 293.948,Z 626.23,A -85,B 0,C 180,E1 -16680.601,E2 -16680.601} C_VEL
LIN {X 0,Y 291.379,Z 614.191,A -85,B 0,C 180,E1 -16684.45,E2 -16684.45} C_VEL
LIN {X 0,Y 291.398,Z 614.185,A -85,B 0,C 180,E1 -16687.259,E2 -16687.259} C_VEL
LIN {X 0,Y 291.377,Z 614.193,A -85,B 0,C 180,E1 -16690.634,E2 -16690.634} C_VEL
LIN {X 0,Y 291.343,Z 614.196,A -85,B 0,C 180,E1 -16694.39,E2 -16694.39} C_VEL
LIN {X 0,Y 291.354,Z 614.193,A -85,B 0,C 180,E1 -16698.397,E2 -16698.397} C_VEL
LIN {X 0,Y 291.373,Z 614.19,A -85,B 0,C 180,E1 -16701.161,E2 -16701.161} C_VEL
LIN {X 0,Y 291.383,Z 614.19,A -85,B 0,C 180,E1 -16704.628,E2 -16704.628} C_VEL
LIN {X 0,Y 291.372,Z 614.188,A -85,B 0,C 180,E1 -16707.95,E2 -16707.95} C_VEL
LIN {X 0,Y 291.379,Z 614.19,A -85,B 0,C 180,E1 -16711.157,E2 -16711.157} C_VEL
LIN {X 0,Y 291.411,Z 614.181,A -85,B 0,C 180,E1 -16714.271,E2 -16714.271} C_VEL
LIN {X 0,Y 291.369,Z 614.191,A -85,B 0,C 180,E1 -16717.298,E2 -16717.298} C_VEL
LIN {X 0,Y 291.453,Z 614.177,A -85,B 0,C 180,E1 -16720.269,E2 -16720.269} C_VEL
LIN {X 0,Y 291.535,Z 614.168,A -85,B 0,C 180,E1 -16724.633,E2 -16724.633} C_VEL
LIN {X 0,Y 291.53,Z 614.169,A -85,B 0,C 180,E1 -16728.88,E2 -16728.88} C_VEL
LIN {X 0,Y 291.7,Z 614.147,A -85,B 0,C 180,E1 -16731.688,E2 -16731.688} C_VEL
LIN {X 0,Y 291.623,Z 614.156,A -85,B 0,C 180,E1 -16734.467,E2 -16734.467} C_VEL
LIN {X 0,Y 291.884,Z 614.123,A -85,B 0,C 180,E1 -16738.62,E2 -16738.62} C_VEL
LIN {X 0,Y 291.884,Z 614.124,A -85,B 0,C 180,E1 -16741.379,E2 -16741.379} C_VEL
LIN {X 0,Y 291.736,Z 614.143,A -85,B 0,C 180,E1 -16746.917,E2 -16746.917} C_VEL
LIN {X 0,Y 291.622,Z 614.159,A -85,B 0,C 180,E1 -16749.711,E2 -16749.711} C_VEL
LIN {X 0,Y 291.514,Z 614.17,A -85,B 0,C 180,E1 -16753.95,E2 -16753.95} C_VEL
LIN {X 0,Y 291.479,Z 614.173,A -85,B 0,C 180,E1 -16756.818,E2 -16756.818} C_VEL
LIN {X 0,Y 291.444,Z 614.183,A -85,B 0,C 180,E1 -16759.875,E2 -16759.875} C_VEL
LIN {X 0,Y 291.393,Z 614.183,A -85,B 0,C 180,E1 -16764.205,E2 -16764.205} C_VEL
LIN {X 0,Y 291.415,Z 614.179,A -85,B 0,C 180,E1 -16767.271,E2 -16767.271} C_VEL
LIN {X 0,Y 291.332,Z 614.194,A -85,B 0,C 180,E1 -16770.437,E2 -16770.437} C_VEL
LIN {X 0,Y 291.338,Z 614.193,A -85,B 0,C 180,E1 -16773.698,E2 -16773.698} C_VEL
LIN {X 0,Y 291.397,Z 614.18,A -85,B 0,C 180,E1 -16777.261,E2 -16777.261} C_VEL
LIN {X 0,Y 291.395,Z 614.185,A -85,B 0,C 180,E1 -16780.631,E2 -16780.631} C_VEL
LIN {X 0,Y 291.348,Z 614.194,A -85,B 0,C 180,E1 -16784.39,E2 -16784.39} C_VEL
LIN {X 0,Y 291.351,Z 614.191,A -85,B 0,C 180,E1 -16788.398,E2 -16788.398} C_VEL
LIN {X 0,Y 291.368,Z 614.186,A -85,B 0,C 180,E1 -16791.162,E2 -16791.162} C_VEL
LIN {X 0,Y 291.38,Z 614.19,A -85,B 0,C 180,E1 -16794.63,E2 -16794.63} C_VEL
LIN {X 0,Y 291.365,Z 614.188,A -85,B 0,C 180,E1 -16797.951,E2 -16797.951} C_VEL
LIN {X 0,Y 291.372,Z 614.188,A -85,B 0,C 180,E1 -16801.158,E2 -16801.158} C_VEL
LIN {X 0,Y 291.408,Z 614.185,A -85,B 0,C 180,E1 -16804.272,E2 -16804.272} C_VEL
LIN {X 0,Y 291.378,Z 614.188,A -85,B 0,C 180,E1 -16807.3,E2 -16807.3} C_VEL
LIN {X 0,Y 291.454,Z 614.178,A -85,B 0,C 180,E1 -16810.27,E2 -16810.27} C_VEL
LIN {X 0,Y 291.552,Z 614.168,A -85,B 0,C 180,E1 -16814.624,E2 -16814.624} C_VEL
LIN {X 0,Y 291.533,Z 614.171,A -85,B 0,C 180,E1 -16818.881,E2 -16818.881} C_VEL
LIN {X 0,Y 291.702,Z 614.145,A -85,B 0,C 180,E1 -16821.689,E2 -16821.689} C_VEL
LIN {X 0,Y 291.626,Z 614.156,A -85,B 0,C 180,E1 -16824.468,E2 -16824.468} C_VEL
LIN {X 0,Y 291.887,Z 614.124,A -85,B 0,C 180,E1 -16828.62,E2 -16828.62} C_VEL
LIN {X 0,Y 291.887,Z 614.126,A -85,B 0,C 180,E1 -16831.38,E2 -16831.38} C_VEL
LIN {X 0,Y 291.732,Z 614.146,A -85,B 0,C 180,E1 -16836.918,E2 -16836.918} C_VEL
LIN {X 0,Y 291.572,Z 614.165,A -85,B 0,C 180,E1 -16839.714,E2 -16839.714} C_VEL
LIN {X 0,Y 291.519,Z 614.172,A -85,B 0,C 180,E1 -16843.95,E2 -16843.95} C_VEL
LIN {X 0,Y 291.486,Z 614.176,A -85,B 0,C 180,E1 -16846.817,E2 -16846.817} C_VEL
LIN {X 0,Y 291.502,Z 614.215,A -85,B 0,C 180,E1 -16848.447,E2 -16848.447} C_VEL
LIN {X 0,Y 291.543,Z 614.456,A -85,B 0,C 180,E1 -16848.536,E2 -16848.536} C_VEL
LIN {X 0,Y 302.827,Z 645.282,A -85,B 0,C 180,E1 -16850.302,E2 -16850.302} C_VEL
LIN {X 0,Y 300.517,Z 722.156,A -85,B 0,C 180,E1 -16852.335,E2 -16852.335} C_VEL
LIN {X 0,Y 299.797,Z 735.876,A -85,B 0,C 180,E1 -16852.983,E2 -16852.983} C_VEL
LIN {X 0,Y 298.864,Z 748.524,A -85,B 0,C 180,E1 -16853.861,E2 -16853.861} C_VEL
LIN {X 0,Y 297.636,Z 761.17,A -85,B 0,C 180,E1 -16855.049,E2 -16855.049} C_VEL
LIN {X 0,Y 296.392,Z 771.663,A -85,B 0,C 180,E1 -16856.306,E2 -16856.306} C_VEL
LIN {X 0,Y 295.01,Z 782.234,A -85,B 0,C 180,E1 -16857.895,E2 -16857.895} C_VEL
LIN {X 0,Y 293.691,Z 792.189,A -85,B 0,C 180,E1 -16859.771,E2 -16859.771} C_VEL
LIN {X 0,Y 292.591,Z 799.711,A -85,B 0,C 180,E1 -16861.513,E2 -16861.513} C_VEL
LIN {X 0,Y 291.52,Z 807.24,A -85,B 0,C 180,E1 -16863.674,E2 -16863.674} C_VEL
LIN {X 0,Y 290.838,Z 812.218,A -85,B 0,C 180,E1 -16865.446,E2 -16865.446} C_VEL
LIN {X 0,Y 290.342,Z 816.282,A -85,B 0,C 180,E1 -16867.238,E2 -16867.238} C_VEL
LIN {X 0,Y 289.715,Z 820.95,A -85,B 0,C 180,E1 -16870.002,E2 -16870.002} C_VEL
LIN {X 0,Y 289.573,Z 822.418,A -85,B 0,C 180,E1 -16871.204,E2 -16871.204} C_VEL
LIN {X 0,Y 289.341,Z 824.176,A -85,B 0,C 180,E1 -16873.224,E2 -16873.224} C_VEL
LIN {X 0,Y 289.287,Z 825.068,A -85,B 0,C 180,E1 -16875.209,E2 -16875.209} C_VEL
LIN {X 0,Y 289.392,Z 825.138,A -85,B 0,C 180,E1 -16877.158,E2 -16877.158} C_VEL
LIN {X 0,Y 289.701,Z 824.397,A -85,B 0,C 180,E1 -16879.081,E2 -16879.081} C_VEL
LIN {X 0,Y 290.103,Z 822.939,A -85,B 0,C 180,E1 -16880.96,E2 -16880.96} C_VEL
LIN {X 0,Y 290.653,Z 820.591,A -85,B 0,C 180,E1 -16882.932,E2 -16882.932} C_VEL
LIN {X 0,Y 291.454,Z 817.004,A -85,B 0,C 180,E1 -16885.069,E2 -16885.069} C_VEL
LIN {X 0,Y 292.51,Z 812.146,A -85,B 0,C 180,E1 -16887.236,E2 -16887.236} C_VEL
LIN {X 0,Y 293.932,Z 805.871,A -85,B 0,C 180,E1 -16889.401,E2 -16889.401} C_VEL
LIN {X 0,Y 295.685,Z 797.892,A -85,B 0,C 180,E1 -16891.572,E2 -16891.572} C_VEL
LIN {X 0,Y 297.634,Z 788.349,A -85,B 0,C 180,E1 -16893.602,E2 -16893.602} C_VEL
LIN {X 0,Y 299.518,Z 778.448,A -85,B 0,C 180,E1 -16895.282,E2 -16895.282} C_VEL
LIN {X 0,Y 301.434,Z 766.845,A -85,B 0,C 180,E1 -16896.827,E2 -16896.827} C_VEL
LIN {X 0,Y 303.122,Z 755.241,A -85,B 0,C 180,E1 -16898.032,E2 -16898.032} C_VEL
LIN {X 0,Y 304.412,Z 743.845,A -85,B 0,C 180,E1 -16898.944,E2 -16898.944} C_VEL
LIN {X 0,Y 305.17,Z 733.808,A -85,B 0,C 180,E1 -16899.565,E2 -16899.565} C_VEL
LIN {X 0,Y 304.814,Z 728.206,A -85,B 0,C 180,E1 -16899.925,E2 -16899.925} C_VEL
LIN {X 0,Y 301.212,Z 711.625,A -85,B 0,C 180,E1 -16900.968,E2 -16900.968} C_VEL
LIN {X 0,Y 300.647,Z 705.894,A -85,B 0,C 180,E1 -16901.21,E2 -16901.21} C_VEL
LIN {X 0,Y 300.675,Z 703.952,A -85,B 0,C 180,E1 -16901.269,E2 -16901.269} C_VEL
LIN {X 0,Y 302.804,Z 653.194,A -85,B 0,C 180,E1 -16902.657,E2 -16902.657} C_VEL
LIN {X 0,Y 296.675,Z 639.171,A -85,B 0,C 180,E1 -16903.952,E2 -16903.952} C_VEL
LIN {X 0,Y 289.61,Z 625.795,A -85,B 0,C 180,E1 -16905.472,E2 -16905.472} C_VEL
LIN {X 0,Y 285.261,Z 618.214,A -85,B 0,C 180,E1 -16906.465,E2 -16906.465} C_VEL
LIN {X 0,Y 284.457,Z 615.055,A -85,B 0,C 180,E1 -16908.149,E2 -16908.149} C_VEL
LIN {X 0,Y 284.653,Z 615.031,A -85,B 0,C 180,E1 -16911.482,E2 -16911.482} C_VEL
LIN {X 0,Y 284.599,Z 615.033,A -85,B 0,C 180,E1 -16914.332,E2 -16914.332} C_VEL
LIN {X 0,Y 284.854,Z 615,A -85,B 0,C 180,E1 -16918.587,E2 -16918.587} C_VEL
LIN {X 0,Y 284.853,Z 614.999,A -85,B 0,C 180,E1 -16921.414,E2 -16921.414} C_VEL
LIN {X 0,Y 284.693,Z 615.018,A -85,B 0,C 180,E1 -16927.091,E2 -16927.091} C_VEL
LIN {X 0,Y 284.561,Z 615.032,A -85,B 0,C 180,E1 -16929.956,E2 -16929.956} C_VEL
LIN {X 0,Y 284.473,Z 615.049,A -85,B 0,C 180,E1 -16934.304,E2 -16934.304} C_VEL
LIN {X 0,Y 284.42,Z 615.056,A -85,B 0,C 180,E1 -16937.249,E2 -16937.249} C_VEL
LIN {X 0,Y 284.374,Z 615.06,A -85,B 0,C 180,E1 -16940.243,E2 -16940.243} C_VEL
LIN {X 0,Y 284.365,Z 615.063,A -85,B 0,C 180,E1 -16943.876,E2 -16943.876} C_VEL
LIN {X 0,Y 284.393,Z 615.057,A -85,B 0,C 180,E1 -16947.175,E2 -16947.175} C_VEL
LIN {X 0,Y 284.295,Z 615.065,A -85,B 0,C 180,E1 -16951.275,E2 -16951.275} C_VEL
LIN {X 0,Y 284.359,Z 615.056,A -85,B 0,C 180,E1 -16955.355,E2 -16955.355} C_VEL
LIN {X 0,Y 284.326,Z 615.061,A -85,B 0,C 180,E1 -16958.168,E2 -16958.168} C_VEL
LIN {X 0,Y 284.3,Z 615.071,A -85,B 0,C 180,E1 -16961.871,E2 -16961.871} C_VEL
LIN {X 0,Y 284.317,Z 615.067,A -85,B 0,C 180,E1 -16966.202,E2 -16966.202} C_VEL
LIN {X 0,Y 284.349,Z 615.138,A -85,B 0,C 180,E1 -16970.076,E2 -16970.076} C_VEL
LIN {X 0,Y 286.479,Z 622.776,A -85,B 0,C 180,E1 -16973.495,E2 -16973.495} C_VEL
LIN {X 0,Y 288.489,Z 630.973,A -85,B 0,C 180,E1 -16976.798,E2 -16976.798} C_VEL
LIN {X 0,Y 289.985,Z 637.824,A -85,B 0,C 180,E1 -16979.308,E2 -16979.308} C_VEL
LIN {X 0,Y 295.955,Z 651.222,A -85,B 0,C 180,E1 -16980.653,E2 -16980.653} C_VEL
LIN {X 0,Y 299.667,Z 671.71,A -85,B 0,C 180,E1 -16981.842,E2 -16981.842} C_VEL
LIN {X 0,Y 301.586,Z 687.723,A -85,B 0,C 180,E1 -16982.607,E2 -16982.607} C_VEL
LIN {X 0,Y 299.555,Z 741.438,A -85,B 0,C 180,E1 -16984.09,E2 -16984.09} C_VEL
LIN {X 0,Y 298.688,Z 754.587,A -85,B 0,C 180,E1 -16984.57,E2 -16984.57} C_VEL
LIN {X 0,Y 297.241,Z 767.489,A -85,B 0,C 180,E1 -16985.279,E2 -16985.279} C_VEL
LIN {X 0,Y 295.681,Z 779.054,A -85,B 0,C 180,E1 -16986.168,E2 -16986.168} C_VEL
LIN {X 0,Y 293.817,Z 790.435,A -85,B 0,C 180,E1 -16987.313,E2 -16987.313} C_VEL
LIN {X 0,Y 291.67,Z 802.065,A -85,B 0,C 180,E1 -16988.812,E2 -16988.812} C_VEL
LIN {X 0,Y 289.578,Z 812.448,A -85,B 0,C 180,E1 -16990.506,E2 -16990.506} C_VEL
LIN {X 0,Y 287.869,Z 820.81,A -85,B 0,C 180,E1 -16992.204,E2 -16992.204} C_VEL
LIN {X 0,Y 286.123,Z 829.258,A -85,B 0,C 180,E1 -16994.325,E2 -16994.325} C_VEL
LIN {X 0,Y 284.665,Z 836.01,A -85,B 0,C 180,E1 -16996.436,E2 -16996.436} C_VEL
LIN {X 0,Y 283.616,Z 841.434,A -85,B 0,C 180,E1 -16998.566,E2 -16998.566} C_VEL
LIN {X 0,Y 282.94,Z 845.686,A -85,B 0,C 180,E1 -17000.709,E2 -17000.709} C_VEL
LIN {X 0,Y 282.573,Z 848.873,A -85,B 0,C 180,E1 -17002.857,E2 -17002.857} C_VEL
LIN {X 0,Y 282.419,Z 850.648,A -85,B 0,C 180,E1 -17004.508,E2 -17004.508} C_VEL
LIN {X 0,Y 282.446,Z 852.335,A -85,B 0,C 180,E1 -17007.148,E2 -17007.148} C_VEL
LIN {X 0,Y 282.44,Z 852.674,A -85,B 0,C 180,E1 -17008.574,E2 -17008.574} C_VEL
LIN {X 0,Y 282.522,Z 852.59,A -85,B 0,C 180,E1 -17010,E2 -17010} C_VEL
LIN {X 0,Y 282.463,Z 852.055,A -85,B 0,C 180,E1 -17011.426,E2 -17011.426} C_VEL
LIN {X 0,Y 282.459,Z 851.115,A -85,B 0,C 180,E1 -17012.852,E2 -17012.852} C_VEL
LIN {X 0,Y 282.453,Z 849.76,A -85,B 0,C 180,E1 -17014.281,E2 -17014.281} C_VEL
LIN {X 0,Y 282.503,Z 846.84,A -85,B 0,C 180,E1 -17016.428,E2 -17016.428} C_VEL
LIN {X 0,Y 282.787,Z 842.841,A -85,B 0,C 180,E1 -17018.575,E2 -17018.575} C_VEL
LIN {X 0,Y 283.386,Z 836.628,A -85,B 0,C 180,E1 -17021.081,E2 -17021.081} C_VEL
LIN {X 0,Y 284.286,Z 829.811,A -85,B 0,C 180,E1 -17023.219,E2 -17023.219} C_VEL
LIN {X 0,Y 285.509,Z 821.327,A -85,B 0,C 180,E1 -17025.344,E2 -17025.344} C_VEL
LIN {X 0,Y 286.638,Z 812.539,A -85,B 0,C 180,E1 -17027.111,E2 -17027.111} C_VEL
LIN {X 0,Y 288.17,Z 801.744,A -85,B 0,C 180,E1 -17028.853,E2 -17028.853} C_VEL
LIN {X 0,Y 289.627,Z 791.04,A -85,B 0,C 180,E1 -17030.229,E2 -17030.229} C_VEL
LIN {X 0,Y 291.055,Z 779.111,A -85,B 0,C 180,E1 -17031.42,E2 -17031.42} C_VEL
LIN {X 0,Y 292.306,Z 766.834,A -85,B 0,C 180,E1 -17032.345,E2 -17032.345} C_VEL
LIN {X 0,Y 293.292,Z 754.455,A -85,B 0,C 180,E1 -17033.009,E2 -17033.009} C_VEL
LIN {X 0,Y 293.899,Z 738.953,A -85,B 0,C 180,E1 -17033.518,E2 -17033.518} C_VEL
LIN {X 0,Y 295.31,Z 685.881,A -85,B 0,C 180,E1 -17034.946,E2 -17034.946} C_VEL
LIN {X 0,Y 289.156,Z 640.573,A -85,B 0,C 180,E1 -17036.776,E2 -17036.776} C_VEL
LIN {X 0,Y 289.154,Z 638.071,A -85,B 0,C 180,E1 -17037.503,E2 -17037.503} C_VEL
LIN {X 0,Y 286.881,Z 626.957,A -85,B 0,C 180,E1 -17040.97,E2 -17040.97} C_VEL
LIN {X 0,Y 284.344,Z 615.065,A -85,B 0,C 180,E1 -17044.91,E2 -17044.91} C_VEL
LIN {X 0,Y 284.33,Z 615.067,A -85,B 0,C 180,E1 -17048.165,E2 -17048.165} C_VEL
LIN {X 0,Y 284.302,Z 615.07,A -85,B 0,C 180,E1 -17051.869,E2 -17051.869} C_VEL
LIN {X 0,Y 284.293,Z 615.071,A -85,B 0,C 180,E1 -17055.798,E2 -17055.798} C_VEL
LIN {X 0,Y 284.35,Z 615.063,A -85,B 0,C 180,E1 -17060.012,E2 -17060.012} C_VEL
LIN {X 0,Y 284.35,Z 615.063,A -85,B 0,C 180,E1 -17063.616,E2 -17063.616} C_VEL
LIN {X 0,Y 284.306,Z 615.07,A -85,B 0,C 180,E1 -17067.188,E2 -17067.188} C_VEL
LIN {X 0,Y 284.356,Z 615.062,A -85,B 0,C 180,E1 -17070.375,E2 -17070.375} C_VEL
LIN {X 0,Y 284.374,Z 615.058,A -85,B 0,C 180,E1 -17073.585,E2 -17073.585} C_VEL
LIN {X 0,Y 284.328,Z 615.067,A -85,B 0,C 180,E1 -17076.703,E2 -17076.703} C_VEL
LIN {X 0,Y 284.394,Z 615.059,A -85,B 0,C 180,E1 -17081.26,E2 -17081.26} C_VEL
LIN {X 0,Y 284.473,Z 615.047,A -85,B 0,C 180,E1 -17084.469,E2 -17084.469} C_VEL
LIN {X 0,Y 284.482,Z 615.046,A -85,B 0,C 180,E1 -17088.601,E2 -17088.601} C_VEL
LIN {X 0,Y 284.651,Z 615.027,A -85,B 0,C 180,E1 -17091.48,E2 -17091.48} C_VEL
LIN {X 0,Y 284.594,Z 615.032,A -85,B 0,C 180,E1 -17094.33,E2 -17094.33} C_VEL
LIN {X 0,Y 284.85,Z 614.999,A -85,B 0,C 180,E1 -17098.586,E2 -17098.586} C_VEL
LIN {X 0,Y 284.85,Z 614.999,A -85,B 0,C 180,E1 -17101.413,E2 -17101.413} C_VEL
LIN {X 0,Y 284.688,Z 615.021,A -85,B 0,C 180,E1 -17107.09,E2 -17107.09} C_VEL
LIN {X 0,Y 284.559,Z 615.036,A -85,B 0,C 180,E1 -17109.955,E2 -17109.955} C_VEL
LIN {X 0,Y 284.47,Z 615.044,A -85,B 0,C 180,E1 -17114.303,E2 -17114.303} C_VEL
LIN {X 0,Y 284.417,Z 615.053,A -85,B 0,C 180,E1 -17117.248,E2 -17117.248} C_VEL
LIN {X 0,Y 284.372,Z 615.06,A -85,B 0,C 180,E1 -17120.242,E2 -17120.242} C_VEL
LIN {X 0,Y 284.362,Z 615.061,A -85,B 0,C 180,E1 -17123.875,E2 -17123.875} C_VEL
LIN {X 0,Y 284.39,Z 615.053,A -85,B 0,C 180,E1 -17127.173,E2 -17127.173} C_VEL
LIN {X 0,Y 284.291,Z 615.069,A -85,B 0,C 180,E1 -17131.274,E2 -17131.274} C_VEL
LIN {X 0,Y 284.355,Z 615.06,A -85,B 0,C 180,E1 -17135.354,E2 -17135.354} C_VEL
LIN {X 0,Y 284.329,Z 615.064,A -85,B 0,C 180,E1 -17138.165,E2 -17138.165} C_VEL
LIN {X 0,Y 284.335,Z 615.068,A -85,B 0,C 180,E1 -17142.141,E2 -17142.141} C_VEL
LIN {X 0,Y 284.313,Z 615.071,A -85,B 0,C 180,E1 -17146.202,E2 -17146.202} C_VEL
LIN {X 0,Y 284.346,Z 615.06,A -85,B 0,C 180,E1 -17150.013,E2 -17150.013} C_VEL
LIN {X 0,Y 284.346,Z 615.063,A -85,B 0,C 180,E1 -17153.617,E2 -17153.617} C_VEL
LIN {X 0,Y 284.302,Z 615.067,A -85,B 0,C 180,E1 -17157.19,E2 -17157.19} C_VEL
LIN {X 0,Y 284.35,Z 615.062,A -85,B 0,C 180,E1 -17160.376,E2 -17160.376} C_VEL
LIN {X 0,Y 284.37,Z 615.06,A -85,B 0,C 180,E1 -17163.587,E2 -17163.587} C_VEL
LIN {X 0,Y 284.362,Z 615.066,A -85,B 0,C 180,E1 -17166.707,E2 -17166.707} C_VEL
LIN {X 0,Y 284.4,Z 615.057,A -85,B 0,C 180,E1 -17171.262,E2 -17171.262} C_VEL
LIN {X 0,Y 284.488,Z 615.047,A -85,B 0,C 180,E1 -17174.459,E2 -17174.459} C_VEL
LIN {X 0,Y 284.485,Z 615.048,A -85,B 0,C 180,E1 -17178.602,E2 -17178.602} C_VEL
LIN {X 0,Y 284.653,Z 615.024,A -85,B 0,C 180,E1 -17181.481,E2 -17181.481} C_VEL
LIN {X 0,Y 284.596,Z 615.031,A -85,B 0,C 180,E1 -17184.331,E2 -17184.331} C_VEL
LIN {X 0,Y 284.853,Z 615,A -85,B 0,C 180,E1 -17188.586,E2 -17188.586} C_VEL
LIN {X 0,Y 284.853,Z 615.002,A -85,B 0,C 180,E1 -17191.414,E2 -17191.414} C_VEL
LIN {X 0,Y 284.683,Z 615.025,A -85,B 0,C 180,E1 -17197.09,E2 -17197.09} C_VEL
LIN {X 0,Y 284.516,Z 615.043,A -85,B 0,C 180,E1 -17199.957,E2 -17199.957} C_VEL
LIN {X 0,Y 284.478,Z 615.048,A -85,B 0,C 180,E1 -17204.303,E2 -17204.303} C_VEL
LIN {X 0,Y 284.456,Z 615.244,A -85,B 0,C 180,E1 -17207.989,E2 -17207.989} C_VEL
LIN {X 0,Y 294.771,Z 642.886,A -85,B 0,C 180,E1 -17209.642,E2 -17209.642} C_VEL
LIN {X 0,Y 296.258,Z 647.72,A -85,B 0,C 180,E1 -17209.893,E2 -17209.893} C_VEL
LIN {X 0,Y 293.798,Z 722.272,A -85,B 0,C 180,E1 -17211.903,E2 -17211.903} C_VEL
LIN {X 0,Y 293.042,Z 736.041,A -85,B 0,C 180,E1 -17212.564,E2 -17212.564} C_VEL
LIN {X 0,Y 292.162,Z 747.651,A -85,B 0,C 180,E1 -17213.371,E2 -17213.371} C_VEL
LIN {X 0,Y 291.043,Z 759.103,A -85,B 0,C 180,E1 -17214.426,E2 -17214.426} C_VEL
LIN {X 0,Y 289.862,Z 769.781,A -85,B 0,C 180,E1 -17215.683,E2 -17215.683} C_VEL
LIN {X 0,Y 288.418,Z 780.174,A -85,B 0,C 180,E1 -17217.197,E2 -17217.197} C_VEL
LIN {X 0,Y 287.212,Z 789.092,A -85,B 0,C 180,E1 -17218.802,E2 -17218.802} C_VEL
LIN {X 0,Y 285.971,Z 797.567,A -85,B 0,C 180,E1 -17220.667,E2 -17220.667} C_VEL
LIN {X 0,Y 284.746,Z 805.81,A -85,B 0,C 180,E1 -17222.948,E2 -17222.948} C_VEL
LIN {X 0,Y 283.832,Z 812.245,A -85,B 0,C 180,E1 -17225.204,E2 -17225.204} C_VEL
LIN {X 0,Y 283.203,Z 817.164,A -85,B 0,C 180,E1 -17227.43,E2 -17227.43} C_VEL
LIN {X 0,Y 282.688,Z 820.761,A -85,B 0,C 180,E1 -17229.584,E2 -17229.584} C_VEL
LIN {X 0,Y 282.345,Z 823.728,A -85,B 0,C 180,E1 -17232.226,E2 -17232.226} C_VEL
LIN {X 0,Y 282.215,Z 825.037,A -85,B 0,C 180,E1 -17234.208,E2 -17234.208} C_VEL
LIN {X 0,Y 282.239,Z 825.56,A -85,B 0,C 180,E1 -17236.229,E2 -17236.229} C_VEL
LIN {X 0,Y 282.442,Z 825.229,A -85,B 0,C 180,E1 -17238.285,E2 -17238.285} C_VEL
LIN {X 0,Y 282.864,Z 824.034,A -85,B 0,C 180,E1 -17240.372,E2 -17240.372} C_VEL
LIN {X 0,Y 283.444,Z 821.896,A -85,B 0,C 180,E1 -17242.506,E2 -17242.506} C_VEL
LIN {X 0,Y 284.508,Z 817.467,A -85,B 0,C 180,E1 -17245.379,E2 -17245.379} C_VEL
LIN {X 0,Y 285.669,Z 812.518,A -85,B 0,C 180,E1 -17247.651,E2 -17247.651} C_VEL
LIN {X 0,Y 287.265,Z 805.983,A -85,B 0,C 180,E1 -17249.953,E2 -17249.953} C_VEL
LIN {X 0,Y 288.914,Z 798.892,A -85,B 0,C 180,E1 -17251.931,E2 -17251.931} C_VEL
LIN {X 0,Y 290.839,Z 790.08,A -85,B 0,C 180,E1 -17253.892,E2 -17253.892} C_VEL
LIN {X 0,Y 292.928,Z 779.639,A -85,B 0,C 180,E1 -17255.739,E2 -17255.739} C_VEL
LIN {X 0,Y 294.778,Z 769.194,A -85,B 0,C 180,E1 -17257.206,E2 -17257.206} C_VEL
LIN {X 0,Y 296.708,Z 756.851,A -85,B 0,C 180,E1 -17258.553,E2 -17258.553} C_VEL
LIN {X 0,Y 298.143,Z 745.183,A -85,B 0,C 180,E1 -17259.534,E2 -17259.534} C_VEL
LIN {X 0,Y 299.17,Z 731.902,A -85,B 0,C 180,E1 -17260.359,E2 -17260.359} C_VEL
LIN {X 0,Y 300.088,Z 718.108,A -85,B 0,C 180,E1 -17260.883,E2 -17260.883} C_VEL
LIN {X 0,Y 300.675,Z 703.952,A -85,B 0,C 180,E1 -17261.269,E2 -17261.269} C_VEL
LIN {X 0,Y 300.362,Z 698.162,A -85,B 0,C 180,E1 -17261.494,E2 -17261.494} C_VEL
LIN {X 0,Y 296.268,Z 679.622,A -85,B 0,C 180,E1 -17262.621,E2 -17262.621} C_VEL
LIN {X 0,Y 296.039,Z 673.833,A -85,B 0,C 180,E1 -17262.846,E2 -17262.846} C_VEL
LIN {X 0,Y 296.814,Z 655.141,A -85,B 0,C 180,E1 -17263.381,E2 -17263.381} C_VEL
LIN {X 0,Y 291.296,Z 642.479,A -85,B 0,C 180,E1 -17264.61,E2 -17264.61} C_VEL
LIN {X 0,Y 284.816,Z 630.112,A -85,B 0,C 180,E1 -17266.08,E2 -17266.08} C_VEL
LIN {X 0,Y 280.111,Z 622.275,A -85,B 0,C 180,E1 -17267.181,E2 -17267.181} C_VEL
LIN {X 0,Y 278.155,Z 618.692,A -85,B 0,C 180,E1 -17267.692,E2 -17267.692} C_VEL
LIN {X 0,Y 277.45,Z 615.926,A -85,B 0,C 180,E1 -17269.234,E2 -17269.234} C_VEL
LIN {X 0,Y 277.647,Z 615.901,A -85,B 0,C 180,E1 -17272.73,E2 -17272.73} C_VEL
LIN {X 0,Y 277.82,Z 615.876,A -85,B 0,C 180,E1 -17278.551,E2 -17278.551} C_VEL
LIN {X 0,Y 277.819,Z 615.875,A -85,B 0,C 180,E1 -17281.45,E2 -17281.45} C_VEL
LIN {X 0,Y 277.648,Z 615.896,A -85,B 0,C 180,E1 -17287.272,E2 -17287.272} C_VEL
LIN {X 0,Y 277.502,Z 615.912,A -85,B 0,C 180,E1 -17290.212,E2 -17290.212} C_VEL
LIN {X 0,Y 277.423,Z 615.929,A -85,B 0,C 180,E1 -17294.675,E2 -17294.675} C_VEL
LIN {X 0,Y 277.34,Z 615.932,A -85,B 0,C 180,E1 -17299.235,E2 -17299.235} C_VEL
LIN {X 0,Y 277.315,Z 615.94,A -85,B 0,C 180,E1 -17304.171,E2 -17304.171} C_VEL
LIN {X 0,Y 277.322,Z 615.938,A -85,B 0,C 180,E1 -17307.506,E2 -17307.506} C_VEL
LIN {X 0,Y 277.269,Z 615.943,A -85,B 0,C 180,E1 -17310.483,E2 -17310.483} C_VEL
LIN {X 0,Y 277.252,Z 615.945,A -85,B 0,C 180,E1 -17313.896,E2 -17313.896} C_VEL
LIN {X 0,Y 277.282,Z 615.94,A -85,B 0,C 180,E1 -17317.468,E2 -17317.468} C_VEL
LIN {X 0,Y 277.238,Z 615.946,A -85,B 0,C 180,E1 -17321.232,E2 -17321.232} C_VEL
LIN {X 0,Y 277.245,Z 615.95,A -85,B 0,C 180,E1 -17325.218,E2 -17325.218} C_VEL
LIN {X 0,Y 277.278,Z 616.047,A -85,B 0,C 180,E1 -17328.936,E2 -17328.936} C_VEL
LIN {X 0,Y 279.372,Z 623.332,A -85,B 0,C 180,E1 -17332.413,E2 -17332.413} C_VEL
LIN {X 0,Y 281.457,Z 631.536,A -85,B 0,C 180,E1 -17335.909,E2 -17335.909} C_VEL
LIN {X 0,Y 282.644,Z 637.188,A -85,B 0,C 180,E1 -17338.115,E2 -17338.115} C_VEL
LIN {X 0,Y 284.864,Z 641.749,A -85,B 0,C 180,E1 -17338.655,E2 -17338.655} C_VEL
LIN {X 0,Y 290.451,Z 654.048,A -85,B 0,C 180,E1 -17339.965,E2 -17339.965} C_VEL
LIN {X 0,Y 293.958,Z 674.311,A -85,B 0,C 180,E1 -17341.175,E2 -17341.175} C_VEL
LIN {X 0,Y 295.698,Z 689.402,A -85,B 0,C 180,E1 -17341.918,E2 -17341.918} C_VEL
LIN {X 0,Y 293.094,Z 747.694,A -85,B 0,C 180,E1 -17343.571,E2 -17343.571} C_VEL
LIN {X 0,Y 291.809,Z 761.422,A -85,B 0,C 180,E1 -17344.214,E2 -17344.214} C_VEL
LIN {X 0,Y 290.128,Z 774.384,A -85,B 0,C 180,E1 -17345.11,E2 -17345.11} C_VEL
LIN {X 0,Y 288.126,Z 786.681,A -85,B 0,C 180,E1 -17346.268,E2 -17346.268} C_VEL
LIN {X 0,Y 286.047,Z 797.789,A -85,B 0,C 180,E1 -17347.616,E2 -17347.616} C_VEL
LIN {X 0,Y 283.703,Z 808.862,A -85,B 0,C 180,E1 -17349.329,E2 -17349.329} C_VEL
LIN {X 0,Y 281.747,Z 817.911,A -85,B 0,C 180,E1 -17351.079,E2 -17351.079} C_VEL
LIN {X 0,Y 279.811,Z 826.801,A -85,B 0,C 180,E1 -17353.212,E2 -17353.212} C_VEL
LIN {X 0,Y 278.228,Z 833.934,A -85,B 0,C 180,E1 -17355.369,E2 -17355.369} C_VEL
LIN {X 0,Y 276.906,Z 839.682,A -85,B 0,C 180,E1 -17357.542,E2 -17357.542} C_VEL
LIN {X 0,Y 276.125,Z 844.235,A -85,B 0,C 180,E1 -17359.737,E2 -17359.737} C_VEL
LIN {X 0,Y 275.726,Z 846.661,A -85,B 0,C 180,E1 -17361.203,E2 -17361.203} C_VEL
LIN {X 0,Y 275.505,Z 848.659,A -85,B 0,C 180,E1 -17362.672,E2 -17362.672} C_VEL
LIN {X 0,Y 275.341,Z 850.536,A -85,B 0,C 180,E1 -17364.546,E2 -17364.546} C_VEL
LIN {X 0,Y 275.372,Z 852.024,A -85,B 0,C 180,E1 -17367.074,E2 -17367.074} C_VEL
LIN {X 0,Y 275.361,Z 852.335,A -85,B 0,C 180,E1 -17368.538,E2 -17368.538} C_VEL
LIN {X 0,Y 275.436,Z 852.2,A -85,B 0,C 180,E1 -17370,E2 -17370} C_VEL
LIN {X 0,Y 275.383,Z 851.639,A -85,B 0,C 180,E1 -17371.462,E2 -17371.462} C_VEL
LIN {X 0,Y 275.386,Z 850.673,A -85,B 0,C 180,E1 -17372.926,E2 -17372.926} C_VEL
LIN {X 0,Y 275.384,Z 847.848,A -85,B 0,C 180,E1 -17375.547,E2 -17375.547} C_VEL
LIN {X 0,Y 275.621,Z 843.699,A -85,B 0,C 180,E1 -17378.062,E2 -17378.062} C_VEL
LIN {X 0,Y 276.058,Z 838.836,A -85,B 0,C 180,E1 -17380.265,E2 -17380.265} C_VEL
LIN {X 0,Y 276.782,Z 832.662,A -85,B 0,C 180,E1 -17382.464,E2 -17382.464} C_VEL
LIN {X 0,Y 277.895,Z 824.964,A -85,B 0,C 180,E1 -17384.649,E2 -17384.649} C_VEL
LIN {X 0,Y 279.003,Z 817.345,A -85,B 0,C 180,E1 -17386.401,E2 -17386.401} C_VEL
LIN {X 0,Y 280.419,Z 807.398,A -85,B 0,C 180,E1 -17388.257,E2 -17388.257} C_VEL
LIN {X 0,Y 282.008,Z 796.708,A -85,B 0,C 180,E1 -17389.849,E2 -17389.849} C_VEL
LIN {X 0,Y 283.362,Z 786.417,A -85,B 0,C 180,E1 -17391.077,E2 -17391.077} C_VEL
LIN {X 0,Y 284.788,Z 774.266,A -85,B 0,C 180,E1 -17392.202,E2 -17392.202} C_VEL
LIN {X 0,Y 286.031,Z 760.948,A -85,B 0,C 180,E1 -17393.101,E2 -17393.101} C_VEL
LIN {X 0,Y 286.865,Z 747.708,A -85,B 0,C 180,E1 -17393.699,E2 -17393.699} C_VEL
LIN {X 0,Y 288.68,Z 686.901,A -85,B 0,C 180,E1 -17395.386,E2 -17395.386} C_VEL
LIN {X 0,Y 282.321,Z 640.554,A -85,B 0,C 180,E1 -17397.293,E2 -17397.293} C_VEL
LIN {X 0,Y 280.377,Z 630.445,A -85,B 0,C 180,E1 -17400.452,E2 -17400.452} C_VEL
LIN {X 0,Y 277.976,Z 619.061,A -85,B 0,C 180,E1 -17404.231,E2 -17404.231} C_VEL
LIN {X 0,Y 277.34,Z 615.936,A -85,B 0,C 180,E1 -17405.315,E2 -17405.315} C_VEL
LIN {X 0,Y 277.266,Z 615.947,A -85,B 0,C 180,E1 -17409.322,E2 -17409.322} C_VEL
LIN {X 0,Y 277.241,Z 615.951,A -85,B 0,C 180,E1 -17413.19,E2 -17413.19} C_VEL
LIN {X 0,Y 277.241,Z 615.949,A -85,B 0,C 180,E1 -17417.318,E2 -17417.318} C_VEL
LIN {X 0,Y 277.264,Z 615.95,A -85,B 0,C 180,E1 -17420.676,E2 -17420.676} C_VEL
LIN {X 0,Y 277.302,Z 615.943,A -85,B 0,C 180,E1 -17424.343,E2 -17424.343} C_VEL
LIN {X 0,Y 277.243,Z 615.948,A -85,B 0,C 180,E1 -17427.835,E2 -17427.835} C_VEL
LIN {X 0,Y 277.286,Z 615.945,A -85,B 0,C 180,E1 -17431.211,E2 -17431.211} C_VEL
LIN {X 0,Y 277.305,Z 615.939,A -85,B 0,C 180,E1 -17434.478,E2 -17434.478} C_VEL
LIN {X 0,Y 277.263,Z 615.946,A -85,B 0,C 180,E1 -17437.652,E2 -17437.652} C_VEL
LIN {X 0,Y 277.337,Z 615.937,A -85,B 0,C 180,E1 -17440.765,E2 -17440.765} C_VEL
LIN {X 0,Y 277.423,Z 615.93,A -85,B 0,C 180,E1 -17445.325,E2 -17445.325} C_VEL
LIN {X 0,Y 277.501,Z 615.913,A -85,B 0,C 180,E1 -17449.788,E2 -17449.788} C_VEL
LIN {X 0,Y 277.643,Z 615.897,A -85,B 0,C 180,E1 -17452.728,E2 -17452.728} C_VEL
LIN {X 0,Y 277.816,Z 615.875,A -85,B 0,C 180,E1 -17458.55,E2 -17458.55} C_VEL
LIN {X 0,Y 277.816,Z 615.875,A -85,B 0,C 180,E1 -17461.449,E2 -17461.449} C_VEL
LIN {X 0,Y 277.643,Z 615.9,A -85,B 0,C 180,E1 -17467.27,E2 -17467.27} C_VEL
LIN {X 0,Y 277.5,Z 615.914,A -85,B 0,C 180,E1 -17470.211,E2 -17470.211} C_VEL
LIN {X 0,Y 277.421,Z 615.921,A -85,B 0,C 180,E1 -17474.674,E2 -17474.674} C_VEL
LIN {X 0,Y 277.337,Z 615.936,A -85,B 0,C 180,E1 -17479.234,E2 -17479.234} C_VEL
LIN {X 0,Y 277.312,Z 615.935,A -85,B 0,C 180,E1 -17484.17,E2 -17484.17} C_VEL
LIN {X 0,Y 277.319,Z 615.935,A -85,B 0,C 180,E1 -17487.505,E2 -17487.505} C_VEL
LIN {X 0,Y 277.265,Z 615.946,A -85,B 0,C 180,E1 -17490.481,E2 -17490.481} C_VEL
LIN {X 0,Y 277.248,Z 615.95,A -85,B 0,C 180,E1 -17493.895,E2 -17493.895} C_VEL
LIN {X 0,Y 277.283,Z 615.938,A -85,B 0,C 180,E1 -17497.466,E2 -17497.466} C_VEL
LIN {X 0,Y 277.258,Z 615.944,A -85,B 0,C 180,E1 -17501.227,E2 -17501.227} C_VEL
LIN {X 0,Y 277.245,Z 615.947,A -85,B 0,C 180,E1 -17505.216,E2 -17505.216} C_VEL
LIN {X 0,Y 277.257,Z 615.94,A -85,B 0,C 180,E1 -17509.503,E2 -17509.503} C_VEL
LIN {X 0,Y 277.28,Z 615.947,A -85,B 0,C 180,E1 -17512.534,E2 -17512.534} C_VEL
LIN {X 0,Y 277.249,Z 615.949,A -85,B 0,C 180,E1 -17516.106,E2 -17516.106} C_VEL
LIN {X 0,Y 277.257,Z 615.942,A -85,B 0,C 180,E1 -17519.539,E2 -17519.539} C_VEL
LIN {X 0,Y 277.351,Z 615.937,A -85,B 0,C 180,E1 -17522.864,E2 -17522.864} C_VEL
LIN {X 0,Y 277.324,Z 615.938,A -85,B 0,C 180,E1 -17526.08,E2 -17526.08} C_VEL
LIN {X 0,Y 277.341,Z 615.94,A -85,B 0,C 180,E1 -17530.766,E2 -17530.766} C_VEL
LIN {X 0,Y 277.431,Z 615.924,A -85,B 0,C 180,E1 -17535.326,E2 -17535.326} C_VEL
LIN {X 0,Y 277.503,Z 615.914,A -85,B 0,C 180,E1 -17539.789,E2 -17539.789} C_VEL
LIN {X 0,Y 277.646,Z 615.899,A -85,B 0,C 180,E1 -17542.729,E2 -17542.729} C_VEL
LIN {X 0,Y 277.819,Z 615.876,A -85,B 0,C 180,E1 -17548.55,E2 -17548.55} C_VEL
LIN {X 0,Y 277.819,Z 615.878,A -85,B 0,C 180,E1 -17551.45,E2 -17551.45} C_VEL
LIN {X 0,Y 277.637,Z 615.903,A -85,B 0,C 180,E1 -17557.271,E2 -17557.271} C_VEL
LIN {X 0,Y 277.458,Z 615.922,A -85,B 0,C 180,E1 -17560.213,E2 -17560.213} C_VEL
LIN {X 0,Y 277.431,Z 615.927,A -85,B 0,C 180,E1 -17564.674,E2 -17564.674} C_VEL
LIN {X 0,Y 277.421,Z 616.062,A -85,B 0,C 180,E1 -17567.412,E2 -17567.412} C_VEL
LIN {X 0,Y 279.139,Z 620.538,A -85,B 0,C 180,E1 -17567.702,E2 -17567.702} C_VEL
LIN {X 0,Y 284.382,Z 634.031,A -85,B 0,C 180,E1 -17568.56,E2 -17568.56} C_VEL
LIN {X 0,Y 289.497,Z 648.431,A -85,B 0,C 180,E1 -17569.403,E2 -17569.403} C_VEL
LIN {X 0,Y 287.082,Z 722.208,A -85,B 0,C 180,E1 -17571.445,E2 -17571.445} C_VEL
LIN {X 0,Y 286.31,Z 736.143,A -85,B 0,C 180,E1 -17572.125,E2 -17572.125} C_VEL
LIN {X 0,Y 285.327,Z 748.637,A -85,B 0,C 180,E1 -17573.018,E2 -17573.018} C_VEL
LIN {X 0,Y 284.091,Z 760.786,A -85,B 0,C 180,E1 -17574.193,E2 -17574.193} C_VEL
LIN {X 0,Y 282.703,Z 772.078,A -85,B 0,C 180,E1 -17575.59,E2 -17575.59} C_VEL
LIN {X 0,Y 281.317,Z 782,A -85,B 0,C 180,E1 -17577.124,E2 -17577.124} C_VEL
LIN {X 0,Y 279.973,Z 791.422,A -85,B 0,C 180,E1 -17578.938,E2 -17578.938} C_VEL
LIN {X 0,Y 278.657,Z 799.956,A -85,B 0,C 180,E1 -17580.963,E2 -17580.963} C_VEL
LIN {X 0,Y 277.48,Z 807.798,A -85,B 0,C 180,E1 -17583.3,E2 -17583.3} C_VEL
LIN {X 0,Y 276.565,Z 814.187,A -85,B 0,C 180,E1 -17585.765,E2 -17585.765} C_VEL
LIN {X 0,Y 275.987,Z 818.417,A -85,B 0,C 180,E1 -17587.871,E2 -17587.871} C_VEL
LIN {X 0,Y 275.509,Z 821.754,A -85,B 0,C 180,E1 -17590.07,E2 -17590.07} C_VEL
LIN {X 0,Y 275.248,Z 824.044,A -85,B 0,C 180,E1 -17592.23,E2 -17592.23} C_VEL
LIN {X 0,Y 275.115,Z 825.401,A -85,B 0,C 180,E1 -17594.335,E2 -17594.335} C_VEL
LIN {X 0,Y 275.154,Z 825.918,A -85,B 0,C 180,E1 -17596.4,E2 -17596.4} C_VEL
LIN {X 0,Y 275.373,Z 825.605,A -85,B 0,C 180,E1 -17598.429,E2 -17598.429} C_VEL
LIN {X 0,Y 275.786,Z 824.546,A -85,B 0,C 180,E1 -17600.426,E2 -17600.426} C_VEL
LIN {X 0,Y 276.334,Z 822.783,A -85,B 0,C 180,E1 -17602.383,E2 -17602.383} C_VEL
LIN {X 0,Y 277.376,Z 818.761,A -85,B 0,C 180,E1 -17605.244,E2 -17605.244} C_VEL
LIN {X 0,Y 278.406,Z 814.758,A -85,B 0,C 180,E1 -17607.285,E2 -17607.285} C_VEL
LIN {X 0,Y 279.684,Z 809.64,A -85,B 0,C 180,E1 -17609.341,E2 -17609.341} C_VEL
LIN {X 0,Y 281.575,Z 802.19,A -85,B 0,C 180,E1 -17611.692,E2 -17611.692} C_VEL
LIN {X 0,Y 283.531,Z 794.06,A -85,B 0,C 180,E1 -17613.701,E2 -17613.701} C_VEL
LIN {X 0,Y 285.603,Z 784.691,A -85,B 0,C 180,E1 -17615.569,E2 -17615.569} C_VEL
LIN {X 0,Y 287.629,Z 774.415,A -85,B 0,C 180,E1 -17617.211,E2 -17617.211} C_VEL
LIN {X 0,Y 289.657,Z 762.796,A -85,B 0,C 180,E1 -17618.658,E2 -17618.658} C_VEL
LIN {X 0,Y 291.367,Z 750.927,A -85,B 0,C 180,E1 -17619.809,E2 -17619.809} C_VEL
LIN {X 0,Y 292.744,Z 737.863,A -85,B 0,C 180,E1 -17620.749,E2 -17620.749} C_VEL
LIN {X 0,Y 293.61,Z 725.923,A -85,B 0,C 180,E1 -17621.351,E2 -17621.351} C_VEL
LIN {X 0,Y 295.062,Z 696.212,A -85,B 0,C 180,E1 -17622.22,E2 -17622.22} C_VEL
LIN {X 0,Y 296.039,Z 673.833,A -85,B 0,C 180,E1 -17622.846,E2 -17622.846} C_VEL
LIN {X 0,Y 295.953,Z 669.961,A -85,B 0,C 180,E1 -17622.99,E2 -17622.99} C_VEL
LIN {X 0,Y 294.815,Z 664.411,A -85,B 0,C 180,E1 -17623.337,E2 -17623.337} C_VEL
LIN {X 0,Y 292.859,Z 659.254,A -85,B 0,C 180,E1 -17623.791,E2 -17623.791} C_VEL
LIN {X 0,Y 286.123,Z 646.128,A -85,B 0,C 180,E1 -17625.261,E2 -17625.261} C_VEL
LIN {X 0,Y 279.524,Z 633.427,A -85,B 0,C 180,E1 -17626.842,E2 -17626.842} C_VEL
LIN {X 0,Y 275.129,Z 626.109,A -85,B 0,C 180,E1 -17627.929,E2 -17627.929} C_VEL
LIN {X 0,Y 272.899,Z 622.576,A -85,B 0,C 180,E1 -17628.5,E2 -17628.5} C_VEL
LIN {X 0,Y 271.052,Z 619.212,A -85,B 0,C 180,E1 -17629.033,E2 -17629.033} C_VEL
LIN {X 0,Y 270.534,Z 616.787,A -85,B 0,C 180,E1 -17630.487,E2 -17630.487} C_VEL
LIN {X 0,Y 270.54,Z 616.785,A -85,B 0,C 180,E1 -17634.036,E2 -17634.036} C_VEL
LIN {X 0,Y 270.786,Z 616.752,A -85,B 0,C 180,E1 -17638.514,E2 -17638.514} C_VEL
LIN {X 0,Y 270.784,Z 616.751,A -85,B 0,C 180,E1 -17641.488,E2 -17641.488} C_VEL
LIN {X 0,Y 270.606,Z 616.774,A -85,B 0,C 180,E1 -17647.462,E2 -17647.462} C_VEL
LIN {X 0,Y 270.437,Z 616.794,A -85,B 0,C 180,E1 -17650.482,E2 -17650.482} C_VEL
LIN {X 0,Y 270.391,Z 616.801,A -85,B 0,C 180,E1 -17655.066,E2 -17655.066} C_VEL
LIN {X 0,Y 270.297,Z 616.81,A -85,B 0,C 180,E1 -17659.757,E2 -17659.757} C_VEL
LIN {X 0,Y 270.27,Z 616.818,A -85,B 0,C 180,E1 -17664.587,E2 -17664.587} C_VEL
LIN {X 0,Y 270.267,Z 616.815,A -85,B 0,C 180,E1 -17667.91,E2 -17667.91} C_VEL
LIN {X 0,Y 270.182,Z 616.821,A -85,B 0,C 180,E1 -17671.349,E2 -17671.349} C_VEL
LIN {X 0,Y 270.212,Z 616.817,A -85,B 0,C 180,E1 -17674.905,E2 -17674.905} C_VEL
LIN {X 0,Y 270.221,Z 616.82,A -85,B 0,C 180,E1 -17678.718,E2 -17678.718} C_VEL
LIN {X 0,Y 270.195,Z 616.829,A -85,B 0,C 180,E1 -17682.555,E2 -17682.555} C_VEL
LIN {X 0,Y 270.202,Z 616.828,A -85,B 0,C 180,E1 -17686.744,E2 -17686.744} C_VEL
LIN {X 0,Y 270.203,Z 616.914,A -85,B 0,C 180,E1 -17687.655,E2 -17687.655} C_VEL
LIN {X 0,Y 272.36,Z 624.183,A -85,B 0,C 180,E1 -17691.368,E2 -17691.368} C_VEL
LIN {X 0,Y 274.441,Z 632.318,A -85,B 0,C 180,E1 -17695.033,E2 -17695.033} C_VEL
LIN {X 0,Y 275.473,Z 636.76,A -85,B 0,C 180,E1 -17696.853,E2 -17696.853} C_VEL
LIN {X 0,Y 277.783,Z 641.423,A -85,B 0,C 180,E1 -17697.452,E2 -17697.452} C_VEL
LIN {X 0,Y 284.139,Z 654.957,A -85,B 0,C 180,E1 -17699.038,E2 -17699.038} C_VEL
LIN {X 0,Y 285.341,Z 658.436,A -85,B 0,C 180,E1 -17699.355,E2 -17699.355} C_VEL
LIN {X 0,Y 288.474,Z 677.879,A -85,B 0,C 180,E1 -17700.525,E2 -17700.525} C_VEL
LIN {X 0,Y 289.816,Z 690.432,A -85,B 0,C 180,E1 -17701.159,E2 -17701.159} C_VEL
LIN {X 0,Y 287.076,Z 747.575,A -85,B 0,C 180,E1 -17702.824,E2 -17702.824} C_VEL
LIN {X 0,Y 285.767,Z 761.201,A -85,B 0,C 180,E1 -17703.48,E2 -17703.48} C_VEL
LIN {X 0,Y 284.101,Z 773.621,A -85,B 0,C 180,E1 -17704.348,E2 -17704.348} C_VEL
LIN {X 0,Y 281.994,Z 785.997,A -85,B 0,C 180,E1 -17705.523,E2 -17705.523} C_VEL
LIN {X 0,Y 279.833,Z 797.161,A -85,B 0,C 180,E1 -17706.895,E2 -17706.895} C_VEL
LIN {X 0,Y 277.573,Z 807.318,A -85,B 0,C 180,E1 -17708.462,E2 -17708.462} C_VEL
LIN {X 0,Y 275.412,Z 816.529,A -85,B 0,C 180,E1 -17710.238,E2 -17710.238} C_VEL
LIN {X 0,Y 273.372,Z 825.557,A -85,B 0,C 180,E1 -17712.418,E2 -17712.418} C_VEL
LIN {X 0,Y 271.635,Z 832.884,A -85,B 0,C 180,E1 -17714.622,E2 -17714.622} C_VEL
LIN {X 0,Y 269.953,Z 839.615,A -85,B 0,C 180,E1 -17717.215,E2 -17717.215} C_VEL
LIN {X 0,Y 269.092,Z 844.103,A -85,B 0,C 180,E1 -17719.466,E2 -17719.466} C_VEL
LIN {X 0,Y 268.687,Z 846.501,A -85,B 0,C 180,E1 -17720.971,E2 -17720.971} C_VEL
LIN {X 0,Y 268.423,Z 848.456,A -85,B 0,C 180,E1 -17722.478,E2 -17722.478} C_VEL
LIN {X 0,Y 268.244,Z 850.468,A -85,B 0,C 180,E1 -17724.63,E2 -17724.63} C_VEL
LIN {X 0,Y 268.275,Z 851.713,A -85,B 0,C 180,E1 -17726.997,E2 -17726.997} C_VEL
LIN {X 0,Y 268.283,Z 851.985,A -85,B 0,C 180,E1 -17728.499,E2 -17728.499} C_VEL
LIN {X 0,Y 268.352,Z 851.811,A -85,B 0,C 180,E1 -17730,E2 -17730} C_VEL
LIN {X 0,Y 268.304,Z 851.224,A -85,B 0,C 180,E1 -17731.501,E2 -17731.501} C_VEL
LIN {X 0,Y 268.314,Z 850.231,A -85,B 0,C 180,E1 -17733.003,E2 -17733.003} C_VEL
LIN {X 0,Y 268.29,Z 847.622,A -85,B 0,C 180,E1 -17735.473,E2 -17735.473} C_VEL
LIN {X 0,Y 268.466,Z 844.489,A -85,B 0,C 180,E1 -17737.521,E2 -17737.521} C_VEL
LIN {X 0,Y 268.854,Z 839.967,A -85,B 0,C 180,E1 -17739.783,E2 -17739.783} C_VEL
LIN {X 0,Y 269.464,Z 834.181,A -85,B 0,C 180,E1 -17742.043,E2 -17742.043} C_VEL
LIN {X 0,Y 270.611,Z 826.903,A -85,B 0,C 180,E1 -17744.283,E2 -17744.283} C_VEL
LIN {X 0,Y 271.957,Z 817.809,A -85,B 0,C 180,E1 -17746.514,E2 -17746.514} C_VEL
LIN {X 0,Y 272.998,Z 810.439,A -85,B 0,C 180,E1 -17747.994,E2 -17747.994} C_VEL
LIN {X 0,Y 274.477,Z 800.541,A -85,B 0,C 180,E1 -17749.637,E2 -17749.637} C_VEL
LIN {X 0,Y 276.069,Z 789.687,A -85,B 0,C 180,E1 -17751.074,E2 -17751.074} C_VEL
LIN {X 0,Y 277.538,Z 777.548,A -85,B 0,C 180,E1 -17752.323,E2 -17752.323} C_VEL
LIN {X 0,Y 278.94,Z 765.049,A -85,B 0,C 180,E1 -17753.281,E2 -17753.281} C_VEL
LIN {X 0,Y 279.891,Z 751.938,A -85,B 0,C 180,E1 -17753.982,E2 -17753.982} C_VEL
LIN {X 0,Y 280.627,Z 732.302,A -85,B 0,C 180,E1 -17754.604,E2 -17754.604} C_VEL
LIN {X 0,Y 281.962,Z 687.265,A -85,B 0,C 180,E1 -17755.877,E2 -17755.877} C_VEL
LIN {X 0,Y 276.02,Z 643.118,A -85,B 0,C 180,E1 -17757.74,E2 -17757.74} C_VEL
LIN {X 0,Y 275.095,Z 639.976,A -85,B 0,C 180,E1 -17757.937,E2 -17757.937} C_VEL
LIN {X 0,Y 272.725,Z 628.412,A -85,B 0,C 180,E1 -17761.744,E2 -17761.744} C_VEL
LIN {X 0,Y 270.301,Z 616.814,A -85,B 0,C 180,E1 -17765.803,E2 -17765.803} C_VEL
LIN {X 0,Y 270.223,Z 616.827,A -85,B 0,C 180,E1 -17768.716,E2 -17768.716} C_VEL
LIN {X 0,Y 270.197,Z 616.832,A -85,B 0,C 180,E1 -17772.552,E2 -17772.552} C_VEL
LIN {X 0,Y 270.192,Z 616.831,A -85,B 0,C 180,E1 -17776.744,E2 -17776.744} C_VEL
LIN {X 0,Y 270.235,Z 616.821,A -85,B 0,C 180,E1 -17779.444,E2 -17779.444} C_VEL
LIN {X 0,Y 270.254,Z 616.819,A -85,B 0,C 180,E1 -17783.72,E2 -17783.72} C_VEL
LIN {X 0,Y 270.202,Z 616.83,A -85,B 0,C 180,E1 -17786.892,E2 -17786.892} C_VEL
LIN {X 0,Y 270.226,Z 616.822,A -85,B 0,C 180,E1 -17790.386,E2 -17790.386} C_VEL
LIN {X 0,Y 270.258,Z 616.816,A -85,B 0,C 180,E1 -17793.762,E2 -17793.762} C_VEL
LIN {X 0,Y 270.206,Z 616.829,A -85,B 0,C 180,E1 -17797.036,E2 -17797.036} C_VEL
LIN {X 0,Y 270.295,Z 616.812,A -85,B 0,C 180,E1 -17800.243,E2 -17800.243} C_VEL
LIN {X 0,Y 270.391,Z 616.804,A -85,B 0,C 180,E1 -17804.934,E2 -17804.934} C_VEL
LIN {X 0,Y 270.436,Z 616.794,A -85,B 0,C 180,E1 -17809.518,E2 -17809.518} C_VEL
LIN {X 0,Y 270.602,Z 616.773,A -85,B 0,C 180,E1 -17812.538,E2 -17812.538} C_VEL
LIN {X 0,Y 270.782,Z 616.751,A -85,B 0,C 180,E1 -17818.512,E2 -17818.512} C_VEL
LIN {X 0,Y 270.782,Z 616.75,A -85,B 0,C 180,E1 -17821.486,E2 -17821.486} C_VEL
LIN {X 0,Y 270.602,Z 616.779,A -85,B 0,C 180,E1 -17827.461,E2 -17827.461} C_VEL
LIN {X 0,Y 270.435,Z 616.793,A -85,B 0,C 180,E1 -17830.481,E2 -17830.481} C_VEL
LIN {X 0,Y 270.389,Z 616.797,A -85,B 0,C 180,E1 -17835.065,E2 -17835.065} C_VEL
LIN {X 0,Y 270.294,Z 616.817,A -85,B 0,C 180,E1 -17839.755,E2 -17839.755} C_VEL
LIN {X 0,Y 270.267,Z 616.81,A -85,B 0,C 180,E1 -17844.585,E2 -17844.585} C_VEL
LIN {X 0,Y 270.264,Z 616.816,A -85,B 0,C 180,E1 -17847.909,E2 -17847.909} C_VEL
LIN {X 0,Y 270.178,Z 616.827,A -85,B 0,C 180,E1 -17851.348,E2 -17851.348} C_VEL
LIN {X 0,Y 270.209,Z 616.821,A -85,B 0,C 180,E1 -17854.903,E2 -17854.903} C_VEL
LIN {X 0,Y 270.216,Z 616.819,A -85,B 0,C 180,E1 -17858.717,E2 -17858.717} C_VEL
LIN {X 0,Y 270.216,Z 616.825,A -85,B 0,C 180,E1 -17862.548,E2 -17862.548} C_VEL
LIN {X 0,Y 270.198,Z 616.824,A -85,B 0,C 180,E1 -17866.742,E2 -17866.742} C_VEL
LIN {X 0,Y 270.208,Z 616.818,A -85,B 0,C 180,E1 -17869.442,E2 -17869.442} C_VEL
LIN {X 0,Y 270.251,Z 616.819,A -85,B 0,C 180,E1 -17873.722,E2 -17873.722} C_VEL
LIN {X 0,Y 270.199,Z 616.825,A -85,B 0,C 180,E1 -17876.893,E2 -17876.893} C_VEL
LIN {X 0,Y 270.19,Z 616.825,A -85,B 0,C 180,E1 -17880.383,E2 -17880.383} C_VEL
LIN {X 0,Y 270.257,Z 616.818,A -85,B 0,C 180,E1 -17883.764,E2 -17883.764} C_VEL
LIN {X 0,Y 270.229,Z 616.824,A -85,B 0,C 180,E1 -17887.039,E2 -17887.039} C_VEL
LIN {X 0,Y 270.298,Z 616.814,A -85,B 0,C 180,E1 -17890.245,E2 -17890.245} C_VEL
LIN {X 0,Y 270.4,Z 616.803,A -85,B 0,C 180,E1 -17894.936,E2 -17894.936} C_VEL
LIN {X 0,Y 270.438,Z 616.795,A -85,B 0,C 180,E1 -17899.519,E2 -17899.519} C_VEL
LIN {X 0,Y 270.604,Z 616.775,A -85,B 0,C 180,E1 -17902.539,E2 -17902.539} C_VEL
LIN {X 0,Y 270.785,Z 616.752,A -85,B 0,C 180,E1 -17908.513,E2 -17908.513} C_VEL
LIN {X 0,Y 270.785,Z 616.753,A -85,B 0,C 180,E1 -17911.487,E2 -17911.487} C_VEL
LIN {X 0,Y 270.595,Z 616.779,A -85,B 0,C 180,E1 -17917.461,E2 -17917.461} C_VEL
LIN {X 0,Y 270.41,Z 616.8,A -85,B 0,C 180,E1 -17920.482,E2 -17920.482} C_VEL
LIN {X 0,Y 270.4,Z 616.805,A -85,B 0,C 180,E1 -17925.064,E2 -17925.064} C_VEL
LIN {X 0,Y 270.362,Z 616.877,A -85,B 0,C 180,E1 -17926.809,E2 -17926.809} C_VEL
LIN {X 0,Y 272.209,Z 621.676,A -85,B 0,C 180,E1 -17927.132,E2 -17927.132} C_VEL
LIN {X 0,Y 276.276,Z 631.611,A -85,B 0,C 180,E1 -17927.807,E2 -17927.807} C_VEL
LIN {X 0,Y 282.914,Z 650.077,A -85,B 0,C 180,E1 -17928.932,E2 -17928.932} C_VEL
LIN {X 0,Y 280.382,Z 722.398,A -85,B 0,C 180,E1 -17930.977,E2 -17930.977} C_VEL
LIN {X 0,Y 279.595,Z 736.51,A -85,B 0,C 180,E1 -17931.682,E2 -17931.682} C_VEL
LIN {X 0,Y 278.501,Z 749.44,A -85,B 0,C 180,E1 -17932.633,E2 -17932.633} C_VEL
LIN {X 0,Y 277.154,Z 762.37,A -85,B 0,C 180,E1 -17933.936,E2 -17933.936} C_VEL
LIN {X 0,Y 275.852,Z 772.389,A -85,B 0,C 180,E1 -17935.22,E2 -17935.22} C_VEL
LIN {X 0,Y 274.312,Z 783.035,A -85,B 0,C 180,E1 -17936.921,E2 -17936.921} C_VEL
LIN {X 0,Y 272.881,Z 792.783,A -85,B 0,C 180,E1 -17938.878,E2 -17938.878} C_VEL
LIN {X 0,Y 271.667,Z 800.29,A -85,B 0,C 180,E1 -17940.725,E2 -17940.725} C_VEL
LIN {X 0,Y 270.468,Z 807.993,A -85,B 0,C 180,E1 -17943.07,E2 -17943.07} C_VEL
LIN {X 0,Y 269.557,Z 814.207,A -85,B 0,C 180,E1 -17945.505,E2 -17945.505} C_VEL
LIN {X 0,Y 268.964,Z 818.428,A -85,B 0,C 180,E1 -17947.618,E2 -17947.618} C_VEL
LIN {X 0,Y 268.48,Z 821.683,A -85,B 0,C 180,E1 -17949.734,E2 -17949.734} C_VEL
LIN {X 0,Y 268.307,Z 823.087,A -85,B 0,C 180,E1 -17950.907,E2 -17950.907} C_VEL
LIN {X 0,Y 268.092,Z 824.934,A -85,B 0,C 180,E1 -17952.966,E2 -17952.966} C_VEL
LIN {X 0,Y 268.029,Z 825.98,A -85,B 0,C 180,E1 -17955.068,E2 -17955.068} C_VEL
LIN {X 0,Y 268.121,Z 826.243,A -85,B 0,C 180,E1 -17957.216,E2 -17957.216} C_VEL
LIN {X 0,Y 268.463,Z 825.673,A -85,B 0,C 180,E1 -17959.39,E2 -17959.39} C_VEL
LIN {X 0,Y 268.998,Z 824.215,A -85,B 0,C 180,E1 -17961.608,E2 -17961.608} C_VEL
LIN {X 0,Y 269.732,Z 821.772,A -85,B 0,C 180,E1 -17963.872,E2 -17963.872} C_VEL
LIN {X 0,Y 270.732,Z 818.228,A -85,B 0,C 180,E1 -17966.168,E2 -17966.168} C_VEL
LIN {X 0,Y 272.307,Z 812.387,A -85,B 0,C 180,E1 -17968.925,E2 -17968.925} C_VEL
LIN {X 0,Y 274.076,Z 805.867,A -85,B 0,C 180,E1 -17971.263,E2 -17971.263} C_VEL
LIN {X 0,Y 276.154,Z 798.028,A -85,B 0,C 180,E1 -17973.452,E2 -17973.452} C_VEL
LIN {X 0,Y 278.428,Z 788.534,A -85,B 0,C 180,E1 -17975.562,E2 -17975.562} C_VEL
LIN {X 0,Y 280.541,Z 778.908,A -85,B 0,C 180,E1 -17977.259,E2 -17977.259} C_VEL
LIN {X 0,Y 282.446,Z 769.033,A -85,B 0,C 180,E1 -17978.66,E2 -17978.66} C_VEL
LIN {X 0,Y 284.525,Z 756.674,A -85,B 0,C 180,E1 -17980.036,E2 -17980.036} C_VEL
LIN {X 0,Y 286.189,Z 743.908,A -85,B 0,C 180,E1 -17981.105,E2 -17981.105} C_VEL
LIN {X 0,Y 287.24,Z 731.602,A -85,B 0,C 180,E1 -17981.867,E2 -17981.867} C_VEL
LIN {X 0,Y 288.154,Z 718.469,A -85,B 0,C 180,E1 -17982.374,E2 -17982.374} C_VEL
LIN {X 0,Y 291.019,Z 657.283,A -85,B 0,C 180,E1 -17984.125,E2 -17984.125} C_VEL
LIN {X 0,Y 286.123,Z 646.128,A -85,B 0,C 180,E1 -17985.261,E2 -17985.261} C_VEL
LIN {X 0,Y 284.136,Z 643.422,A -85,B 0,C 180,E1 -17985.684,E2 -17985.684} C_VEL
LIN {X 0,Y 279.734,Z 640.467,A -85,B 0,C 180,E1 -17986.53,E2 -17986.53} C_VEL
LIN {X 0,Y 275.322,Z 637.609,A -85,B 0,C 180,E1 -17987.42,E2 -17987.42} C_VEL
LIN {X 0,Y 273.292,Z 635.032,A -85,B 0,C 180,E1 -17987.901,E2 -17987.901} C_VEL
LIN {X 0,Y 268.821,Z 627.721,A -85,B 0,C 180,E1 -17989.083,E2 -17989.083} C_VEL
LIN {X 0,Y 266.301,Z 623.691,A -85,B 0,C 180,E1 -17989.787,E2 -17989.787} C_VEL
LIN {X 0,Y 264.049,Z 619.78,A -85,B 0,C 180,E1 -17990.473,E2 -17990.473} C_VEL
LIN {X 0,Y 263.524,Z 617.661,A -85,B 0,C 180,E1 -17991.856,E2 -17991.856} C_VEL
LIN {X 0,Y 263.388,Z 617.678,A -85,B 0,C 180,E1 -17995.409,E2 -17995.409} C_VEL
LIN {X 0,Y 263.752,Z 617.628,A -85,B 0,C 180,E1 -17998.474,E2 -17998.474} C_VEL
LIN {X 0,Y 263.749,Z 617.627,A -85,B 0,C 180,E1 -18001.528,E2 -18001.528} C_VEL
LIN {X 0,Y 263.568,Z 617.652,A -85,B 0,C 180,E1 -18007.663,E2 -18007.663} C_VEL
LIN {X 0,Y 263.369,Z 617.676,A -85,B 0,C 180,E1 -18010.767,E2 -18010.767} C_VEL
LIN {X 0,Y 263.34,Z 617.676,A -85,B 0,C 180,E1 -18015.479,E2 -18015.479} C_VEL
LIN {X 0,Y 263.259,Z 617.691,A -85,B 0,C 180,E1 -18020.308,E2 -18020.308} C_VEL
LIN {X 0,Y 263.205,Z 617.691,A -85,B 0,C 180,E1 -18025.292,E2 -18025.292} C_VEL
LIN {X 0,Y 263.163,Z 617.694,A -85,B 0,C 180,E1 -18028.732,E2 -18028.732} C_VEL
LIN {X 0,Y 263.131,Z 617.697,A -85,B 0,C 180,E1 -18032.289,E2 -18032.289} C_VEL
LIN {X 0,Y 263.186,Z 617.696,A -85,B 0,C 180,E1 -18035.979,E2 -18035.979} C_VEL
LIN {X 0,Y 263.138,Z 617.706,A -85,B 0,C 180,E1 -18039.867,E2 -18039.867} C_VEL
LIN {X 0,Y 263.138,Z 617.704,A -85,B 0,C 180,E1 -18043.982,E2 -18043.982} C_VEL
LIN {X 0,Y 263.158,Z 617.861,A -85,B 0,C 180,E1 -18046.282,E2 -18046.282} C_VEL
LIN {X 0,Y 265.565,Z 625.7,A -85,B 0,C 180,E1 -18050.571,E2 -18050.571} C_VEL
LIN {X 0,Y 267.677,Z 633.993,A -85,B 0,C 180,E1 -18054.482,E2 -18054.482} C_VEL
LIN {X 0,Y 268.245,Z 636.341,A -85,B 0,C 180,E1 -18055.453,E2 -18055.453} C_VEL
LIN {X 0,Y 270.565,Z 640.837,A -85,B 0,C 180,E1 -18056.1,E2 -18056.1} C_VEL
LIN {X 0,Y 277.328,Z 654.483,A -85,B 0,C 180,E1 -18057.89,E2 -18057.89} C_VEL
LIN {X 0,Y 279.964,Z 661.231,A -85,B 0,C 180,E1 -18058.597,E2 -18058.597} C_VEL
LIN {X 0,Y 282.843,Z 680.013,A -85,B 0,C 180,E1 -18059.77,E2 -18059.77} C_VEL
LIN {X 0,Y 283.978,Z 691.669,A -85,B 0,C 180,E1 -18060.363,E2 -18060.363} C_VEL
LIN {X 0,Y 281.228,Z 746.929,A -85,B 0,C 180,E1 -18062.009,E2 -18062.009} C_VEL
LIN {X 0,Y 279.853,Z 760.554,A -85,B 0,C 180,E1 -18062.672,E2 -18062.672} C_VEL
LIN {X 0,Y 278.084,Z 773.005,A -85,B 0,C 180,E1 -18063.55,E2 -18063.55} C_VEL
LIN {X 0,Y 275.913,Z 785.371,A -85,B 0,C 180,E1 -18064.745,E2 -18064.745} C_VEL
LIN {X 0,Y 273.651,Z 796.535,A -85,B 0,C 180,E1 -18066.141,E2 -18066.141} C_VEL
LIN {X 0,Y 271.261,Z 806.754,A -85,B 0,C 180,E1 -18067.734,E2 -18067.734} C_VEL
LIN {X 0,Y 268.751,Z 816.829,A -85,B 0,C 180,E1 -18069.727,E2 -18069.727} C_VEL
LIN {X 0,Y 266.612,Z 825.755,A -85,B 0,C 180,E1 -18071.957,E2 -18071.957} C_VEL
LIN {X 0,Y 264.792,Z 832.942,A -85,B 0,C 180,E1 -18074.214,E2 -18074.214} C_VEL
LIN {X 0,Y 263.019,Z 839.565,A -85,B 0,C 180,E1 -18076.872,E2 -18076.872} C_VEL
LIN {X 0,Y 262.069,Z 843.975,A -85,B 0,C 180,E1 -18079.18,E2 -18079.18} C_VEL
LIN {X 0,Y 261.664,Z 846.343,A -85,B 0,C 180,E1 -18080.726,E2 -18080.726} C_VEL
LIN {X 0,Y 261.353,Z 848.237,A -85,B 0,C 180,E1 -18082.273,E2 -18082.273} C_VEL
LIN {X 0,Y 261.167,Z 850.341,A -85,B 0,C 180,E1 -18084.673,E2 -18084.673} C_VEL
LIN {X 0,Y 261.182,Z 851.406,A -85,B 0,C 180,E1 -18086.915,E2 -18086.915} C_VEL
LIN {X 0,Y 261.207,Z 851.62,A -85,B 0,C 180,E1 -18088.458,E2 -18088.458} C_VEL
LIN {X 0,Y 261.271,Z 851.414,A -85,B 0,C 180,E1 -18090,E2 -18090} C_VEL
LIN {X 0,Y 261.228,Z 850.799,A -85,B 0,C 180,E1 -18091.542,E2 -18091.542} C_VEL
LIN {X 0,Y 261.243,Z 849.775,A -85,B 0,C 180,E1 -18093.084,E2 -18093.084} C_VEL
LIN {X 0,Y 261.198,Z 847.367,A -85,B 0,C 180,E1 -18095.4,E2 -18095.4} C_VEL
LIN {X 0,Y 261.389,Z 843.906,A -85,B 0,C 180,E1 -18097.726,E2 -18097.726} C_VEL
LIN {X 0,Y 261.802,Z 839.312,A -85,B 0,C 180,E1 -18100.049,E2 -18100.049} C_VEL
LIN {X 0,Y 262.679,Z 832.287,A -85,B 0,C 180,E1 -18102.752,E2 -18102.752} C_VEL
LIN {X 0,Y 263.84,Z 824.65,A -85,B 0,C 180,E1 -18105.053,E2 -18105.053} C_VEL
LIN {X 0,Y 265.006,Z 816.825,A -85,B 0,C 180,E1 -18106.961,E2 -18106.961} C_VEL
LIN {X 0,Y 266.533,Z 807.28,A -85,B 0,C 180,E1 -18108.845,E2 -18108.845} C_VEL
LIN {X 0,Y 268.21,Z 796.702,A -85,B 0,C 180,E1 -18110.516,E2 -18110.516} C_VEL
LIN {X 0,Y 269.887,Z 784.97,A -85,B 0,C 180,E1 -18111.982,E2 -18111.982} C_VEL
LIN {X 0,Y 271.276,Z 773.638,A -85,B 0,C 180,E1 -18113.069,E2 -18113.069} C_VEL
LIN {X 0,Y 272.554,Z 760.348,A -85,B 0,C 180,E1 -18114.011,E2 -18114.011} C_VEL
LIN {X 0,Y 273.436,Z 747.218,A -85,B 0,C 180,E1 -18114.636,E2 -18114.636} C_VEL
LIN {X 0,Y 275.328,Z 687.943,A -85,B 0,C 180,E1 -18116.375,E2 -18116.375} C_VEL
LIN {X 0,Y 269.597,Z 645.105,A -85,B 0,C 180,E1 -18118.229,E2 -18118.229} C_VEL
LIN {X 0,Y 267.773,Z 639.624,A -85,B 0,C 180,E1 -18118.59,E2 -18118.59} C_VEL
LIN {X 0,Y 265.478,Z 628.371,A -85,B 0,C 180,E1 -18122.415,E2 -18122.415} C_VEL
LIN {X 0,Y 263.23,Z 617.697,A -85,B 0,C 180,E1 -18126.267,E2 -18126.267} C_VEL
LIN {X 0,Y 263.154,Z 617.706,A -85,B 0,C 180,E1 -18129.862,E2 -18129.862} C_VEL
LIN {X 0,Y 263.138,Z 617.708,A -85,B 0,C 180,E1 -18133.979,E2 -18133.979} C_VEL
LIN {X 0,Y 263.147,Z 617.707,A -85,B 0,C 180,E1 -18138.399,E2 -18138.399} C_VEL
LIN {X 0,Y 263.186,Z 617.7,A -85,B 0,C 180,E1 -18142.107,E2 -18142.107} C_VEL
LIN {X 0,Y 263.182,Z 617.7,A -85,B 0,C 180,E1 -18145.889,E2 -18145.889} C_VEL
LIN {X 0,Y 263.148,Z 617.704,A -85,B 0,C 180,E1 -18149.506,E2 -18149.506} C_VEL
LIN {X 0,Y 263.189,Z 617.701,A -85,B 0,C 180,E1 -18153.001,E2 -18153.001} C_VEL
LIN {X 0,Y 263.15,Z 617.704,A -85,B 0,C 180,E1 -18156.383,E2 -18156.383} C_VEL
LIN {X 0,Y 263.258,Z 617.69,A -85,B 0,C 180,E1 -18159.692,E2 -18159.692} C_VEL
LIN {X 0,Y 263.34,Z 617.68,A -85,B 0,C 180,E1 -18164.521,E2 -18164.521} C_VEL
LIN {X 0,Y 263.368,Z 617.676,A -85,B 0,C 180,E1 -18169.233,E2 -18169.233} C_VEL
LIN {X 0,Y 263.564,Z 617.649,A -85,B 0,C 180,E1 -18172.337,E2 -18172.337} C_VEL
LIN {X 0,Y 263.746,Z 617.627,A -85,B 0,C 180,E1 -18178.472,E2 -18178.472} C_VEL
LIN {X 0,Y 263.746,Z 617.626,A -85,B 0,C 180,E1 -18181.526,E2 -18181.526} C_VEL
LIN {X 0,Y 263.564,Z 617.655,A -85,B 0,C 180,E1 -18187.661,E2 -18187.661} C_VEL
LIN {X 0,Y 263.367,Z 617.673,A -85,B 0,C 180,E1 -18190.765,E2 -18190.765} C_VEL
LIN {X 0,Y 263.338,Z 617.677,A -85,B 0,C 180,E1 -18195.478,E2 -18195.478} C_VEL
LIN {X 0,Y 263.257,Z 617.69,A -85,B 0,C 180,E1 -18200.306,E2 -18200.306} C_VEL
LIN {X 0,Y 263.202,Z 617.689,A -85,B 0,C 180,E1 -18205.291,E2 -18205.291} C_VEL
LIN {X 0,Y 263.16,Z 617.7,A -85,B 0,C 180,E1 -18208.731,E2 -18208.731} C_VEL
LIN {X 0,Y 263.128,Z 617.708,A -85,B 0,C 180,E1 -18212.288,E2 -18212.288} C_VEL
LIN {X 0,Y 263.184,Z 617.699,A -85,B 0,C 180,E1 -18215.978,E2 -18215.978} C_VEL
LIN {X 0,Y 263.154,Z 617.699,A -85,B 0,C 180,E1 -18219.863,E2 -18219.863} C_VEL
LIN {X 0,Y 263.14,Z 617.707,A -85,B 0,C 180,E1 -18223.979,E2 -18223.979} C_VEL
LIN {X 0,Y 263.152,Z 617.701,A -85,B 0,C 180,E1 -18228.399,E2 -18228.399} C_VEL
LIN {X 0,Y 263.183,Z 617.699,A -85,B 0,C 180,E1 -18232.108,E2 -18232.108} C_VEL
LIN {X 0,Y 263.179,Z 617.701,A -85,B 0,C 180,E1 -18235.891,E2 -18235.891} C_VEL
LIN {X 0,Y 263.136,Z 617.7,A -85,B 0,C 180,E1 -18239.506,E2 -18239.506} C_VEL
LIN {X 0,Y 263.187,Z 617.701,A -85,B 0,C 180,E1 -18243.003,E2 -18243.003} C_VEL
LIN {X 0,Y 263.18,Z 617.701,A -85,B 0,C 180,E1 -18246.387,E2 -18246.387} C_VEL
LIN {X 0,Y 263.26,Z 617.689,A -85,B 0,C 180,E1 -18249.694,E2 -18249.694} C_VEL
LIN {X 0,Y 263.347,Z 617.681,A -85,B 0,C 180,E1 -18254.522,E2 -18254.522} C_VEL
LIN {X 0,Y 263.371,Z 617.676,A -85,B 0,C 180,E1 -18259.235,E2 -18259.235} C_VEL
LIN {X 0,Y 263.566,Z 617.65,A -85,B 0,C 180,E1 -18262.338,E2 -18262.338} C_VEL
LIN {X 0,Y 263.749,Z 617.628,A -85,B 0,C 180,E1 -18268.473,E2 -18268.473} C_VEL
LIN {X 0,Y 263.749,Z 617.63,A -85,B 0,C 180,E1 -18271.527,E2 -18271.527} C_VEL
LIN {X 0,Y 263.555,Z 617.655,A -85,B 0,C 180,E1 -18277.662,E2 -18277.662} C_VEL
LIN {X 0,Y 263.352,Z 617.68,A -85,B 0,C 180,E1 -18280.766,E2 -18280.766} C_VEL
LIN {X 0,Y 263.348,Z 617.684,A -85,B 0,C 180,E1 -18285.478,E2 -18285.478} C_VEL
LIN {X 0,Y 263.325,Z 617.685,A -85,B 0,C 180,E1 -18286.171,E2 -18286.171} C_VEL
LIN {X 0,Y 265.089,Z 622.385,A -85,B 0,C 180,E1 -18286.507,E2 -18286.507} C_VEL
LIN {X 0,Y 269.592,Z 633.046,A -85,B 0,C 180,E1 -18287.273,E2 -18287.273} C_VEL
LIN {X 0,Y 276.229,Z 651.479,A -85,B 0,C 180,E1 -18288.435,E2 -18288.435} C_VEL
LIN {X 0,Y 273.652,Z 723.28,A -85,B 0,C 180,E1 -18290.531,E2 -18290.531} C_VEL
LIN {X 0,Y 272.845,Z 737.19,A -85,B 0,C 180,E1 -18291.253,E2 -18291.253} C_VEL
LIN {X 0,Y 271.754,Z 749.531,A -85,B 0,C 180,E1 -18292.182,E2 -18292.182} C_VEL
LIN {X 0,Y 270.538,Z 760.958,A -85,B 0,C 180,E1 -18293.336,E2 -18293.336} C_VEL
LIN {X 0,Y 269.169,Z 771.578,A -85,B 0,C 180,E1 -18294.693,E2 -18294.693} C_VEL
LIN {X 0,Y 267.653,Z 781.733,A -85,B 0,C 180,E1 -18296.301,E2 -18296.301} C_VEL
LIN {X 0,Y 266.223,Z 791.162,A -85,B 0,C 180,E1 -18298.157,E2 -18298.157} C_VEL
LIN {X 0,Y 264.794,Z 799.854,A -85,B 0,C 180,E1 -18300.283,E2 -18300.283} C_VEL
LIN {X 0,Y 263.522,Z 807.658,A -85,B 0,C 180,E1 -18302.666,E2 -18302.666} C_VEL
LIN {X 0,Y 262.572,Z 813.972,A -85,B 0,C 180,E1 -18305.132,E2 -18305.132} C_VEL
LIN {X 0,Y 261.972,Z 818.234,A -85,B 0,C 180,E1 -18307.245,E2 -18307.245} C_VEL
LIN {X 0,Y 261.302,Z 822.595,A -85,B 0,C 180,E1 -18310.202,E2 -18310.202} C_VEL
LIN {X 0,Y 260.975,Z 825.469,A -85,B 0,C 180,E1 -18313.357,E2 -18313.357} C_VEL
LIN {X 0,Y 260.956,Z 826.451,A -85,B 0,C 180,E1 -18315.556,E2 -18315.556} C_VEL
LIN {X 0,Y 261.079,Z 826.585,A -85,B 0,C 180,E1 -18317.704,E2 -18317.704} C_VEL
LIN {X 0,Y 261.471,Z 825.948,A -85,B 0,C 180,E1 -18319.829,E2 -18319.829} C_VEL
LIN {X 0,Y 261.989,Z 824.597,A -85,B 0,C 180,E1 -18321.905,E2 -18321.905} C_VEL
LIN {X 0,Y 262.667,Z 822.53,A -85,B 0,C 180,E1 -18323.941,E2 -18323.941} C_VEL
LIN {X 0,Y 264.05,Z 818.019,A -85,B 0,C 180,E1 -18326.933,E2 -18326.933} C_VEL
LIN {X 0,Y 265.567,Z 812.795,A -85,B 0,C 180,E1 -18329.429,E2 -18329.429} C_VEL
LIN {X 0,Y 267.389,Z 806.461,A -85,B 0,C 180,E1 -18331.765,E2 -18331.765} C_VEL
LIN {X 0,Y 269.679,Z 798.31,A -85,B 0,C 180,E1 -18334.094,E2 -18334.094} C_VEL
LIN {X 0,Y 272.017,Z 789.063,A -85,B 0,C 180,E1 -18336.191,E2 -18336.191} C_VEL
LIN {X 0,Y 274.199,Z 779.718,A -85,B 0,C 180,E1 -18337.889,E2 -18337.889} C_VEL
LIN {X 0,Y 276.23,Z 769.855,A -85,B 0,C 180,E1 -18339.332,E2 -18339.332} C_VEL
LIN {X 0,Y 278.322,Z 758.102,A -85,B 0,C 180,E1 -18340.688,E2 -18340.688} C_VEL
LIN {X 0,Y 280.046,Z 746.033,A -85,B 0,C 180,E1 -18341.757,E2 -18341.757} C_VEL
LIN {X 0,Y 281.236,Z 733.05,A -85,B 0,C 180,E1 -18342.606,E2 -18342.606} C_VEL
LIN {X 0,Y 282.243,Z 719.866,A -85,B 0,C 180,E1 -18343.142,E2 -18343.142} C_VEL
LIN {X 0,Y 285.263,Z 659.558,A -85,B 0,C 180,E1 -18344.896,E2 -18344.896} C_VEL
LIN {X 0,Y 279.675,Z 646.869,A -85,B 0,C 180,E1 -18346.289,E2 -18346.289} C_VEL
LIN {X 0,Y 273.508,Z 635.421,A -85,B 0,C 180,E1 -18347.844,E2 -18347.844} C_VEL
LIN {X 0,Y 273.292,Z 635.032,A -85,B 0,C 180,E1 -18347.901,E2 -18347.901} C_VEL
LIN {X 0,Y 271.6,Z 632.938,A -85,B 0,C 180,E1 -18348.313,E2 -18348.313} C_VEL
LIN {X 0,Y 268.542,Z 631.196,A -85,B 0,C 180,E1 -18348.995,E2 -18348.995} C_VEL
LIN {X 0,Y 262.334,Z 628.33,A -85,B 0,C 180,E1 -18350.438,E2 -18350.438} C_VEL
LIN {X 0,Y 260.707,Z 626.348,A -85,B 0,C 180,E1 -18350.896,E2 -18350.896} C_VEL
LIN {X 0,Y 260.469,Z 625.843,A -85,B 0,C 180,E1 -18350.974,E2 -18350.974} C_VEL
LIN {X 0,Y 257.233,Z 620.908,A -85,B 0,C 180,E1 -18351.986,E2 -18351.986} C_VEL
LIN {X 0,Y 256.977,Z 620.278,A -85,B 0,C 180,E1 -18352.141,E2 -18352.141} C_VEL
LIN {X 0,Y 256.483,Z 618.54,A -85,B 0,C 180,E1 -18353.412,E2 -18353.412} C_VEL
LIN {X 0,Y 256.717,Z 618.504,A -85,B 0,C 180,E1 -18358.432,E2 -18358.432} C_VEL
LIN {X 0,Y 256.712,Z 618.504,A -85,B 0,C 180,E1 -18361.57,E2 -18361.57} C_VEL
LIN {X 0,Y 256.535,Z 618.53,A -85,B 0,C 180,E1 -18367.874,E2 -18367.874} C_VEL
LIN {X 0,Y 256.305,Z 618.559,A -85,B 0,C 180,E1 -18371.067,E2 -18371.067} C_VEL
LIN {X 0,Y 256.29,Z 618.552,A -85,B 0,C 180,E1 -18375.916,E2 -18375.916} C_VEL
LIN {X 0,Y 256.163,Z 618.578,A -85,B 0,C 180,E1 -18380.896,E2 -18380.896} C_VEL
LIN {X 0,Y 256.185,Z 618.566,A -85,B 0,C 180,E1 -18385.14,E2 -18385.14} C_VEL
LIN {X 0,Y 256.101,Z 618.575,A -85,B 0,C 180,E1 -18389.602,E2 -18389.602} C_VEL
LIN {X 0,Y 256.083,Z 618.581,A -85,B 0,C 180,E1 -18393.291,E2 -18393.291} C_VEL
LIN {X 0,Y 256.137,Z 618.574,A -85,B 0,C 180,E1 -18397.279,E2 -18397.279} C_VEL
LIN {X 0,Y 256.084,Z 618.58,A -85,B 0,C 180,E1 -18401.199,E2 -18401.199} C_VEL
LIN {X 0,Y 256.07,Z 618.644,A -85,B 0,C 180,E1 -18404.64,E2 -18404.64} C_VEL
LIN {X 0,Y 258.207,Z 625.592,A -85,B 0,C 180,E1 -18408.792,E2 -18408.792} C_VEL
LIN {X 0,Y 259.752,Z 631.111,A -85,B 0,C 180,E1 -18411.689,E2 -18411.689} C_VEL
LIN {X 0,Y 260.899,Z 635.701,A -85,B 0,C 180,E1 -18413.864,E2 -18413.864} C_VEL
LIN {X 0,Y 263.433,Z 640.379,A -85,B 0,C 180,E1 -18414.633,E2 -18414.633} C_VEL
LIN {X 0,Y 268.862,Z 650.865,A -85,B 0,C 180,E1 -18416.199,E2 -18416.199} C_VEL
LIN {X 0,Y 274.231,Z 662.677,A -85,B 0,C 180,E1 -18417.681,E2 -18417.681} C_VEL
LIN {X 0,Y 275.543,Z 669.579,A -85,B 0,C 180,E1 -18418.181,E2 -18418.181} C_VEL
LIN {X 0,Y 277.71,Z 685.391,A -85,B 0,C 180,E1 -18419.16,E2 -18419.16} C_VEL
LIN {X 0,Y 278.233,Z 693.069,A -85,B 0,C 180,E1 -18419.539,E2 -18419.539} C_VEL
LIN {X 0,Y 275.428,Z 746.311,A -85,B 0,C 180,E1 -18421.157,E2 -18421.157} C_VEL
LIN {X 0,Y 274.005,Z 759.988,A -85,B 0,C 180,E1 -18421.83,E2 -18421.83} C_VEL
LIN {X 0,Y 272.131,Z 772.5,A -85,B 0,C 180,E1 -18422.716,E2 -18422.716} C_VEL
LIN {X 0,Y 269.887,Z 784.891,A -85,B 0,C 180,E1 -18423.933,E2 -18423.933} C_VEL
LIN {X 0,Y 267.494,Z 796.077,A -85,B 0,C 180,E1 -18425.35,E2 -18425.35} C_VEL
LIN {X 0,Y 265.008,Z 806.274,A -85,B 0,C 180,E1 -18426.973,E2 -18426.973} C_VEL
LIN {X 0,Y 262.579,Z 815.51,A -85,B 0,C 180,E1 -18428.819,E2 -18428.819} C_VEL
LIN {X 0,Y 260.206,Z 824.572,A -85,B 0,C 180,E1 -18431.089,E2 -18431.089} C_VEL
LIN {X 0,Y 258.261,Z 831.943,A -85,B 0,C 180,E1 -18433.398,E2 -18433.398} C_VEL
LIN {X 0,Y 256.565,Z 837.872,A -85,B 0,C 180,E1 -18435.728,E2 -18435.728} C_VEL
LIN {X 0,Y 255.37,Z 842.577,A -85,B 0,C 180,E1 -18438.088,E2 -18438.088} C_VEL
LIN {X 0,Y 254.617,Z 846.194,A -85,B 0,C 180,E1 -18440.467,E2 -18440.467} C_VEL
LIN {X 0,Y 254.307,Z 848.025,A -85,B 0,C 180,E1 -18442.058,E2 -18442.058} C_VEL
LIN {X 0,Y 254.088,Z 850.176,A -85,B 0,C 180,E1 -18444.723,E2 -18444.723} C_VEL
LIN {X 0,Y 254.093,Z 851.086,A -85,B 0,C 180,E1 -18446.829,E2 -18446.829} C_VEL
LIN {X 0,Y 254.132,Z 851.253,A -85,B 0,C 180,E1 -18448.415,E2 -18448.415} C_VEL
LIN {X 0,Y 254.192,Z 851.018,A -85,B 0,C 180,E1 -18450,E2 -18450} C_VEL
LIN {X 0,Y 254.154,Z 850.372,A -85,B 0,C 180,E1 -18451.585,E2 -18451.585} C_VEL
LIN {X 0,Y 254.15,Z 849.294,A -85,B 0,C 180,E1 -18453.17,E2 -18453.17} C_VEL
LIN {X 0,Y 254.128,Z 847.041,A -85,B 0,C 180,E1 -18455.375,E2 -18455.375} C_VEL
LIN {X 0,Y 254.334,Z 843.297,A -85,B 0,C 180,E1 -18457.941,E2 -18457.941} C_VEL
LIN {X 0,Y 254.766,Z 838.609,A -85,B 0,C 180,E1 -18460.329,E2 -18460.329} C_VEL
LIN {X 0,Y 255.519,Z 832.617,A -85,B 0,C 180,E1 -18462.711,E2 -18462.711} C_VEL
LIN {X 0,Y 256.732,Z 825.126,A -85,B 0,C 180,E1 -18465.073,E2 -18465.073} C_VEL
LIN {X 0,Y 257.928,Z 817.464,A -85,B 0,C 180,E1 -18467.032,E2 -18467.032} C_VEL
LIN {X 0,Y 259.434,Z 808.182,A -85,B 0,C 180,E1 -18468.97,E2 -18468.97} C_VEL
LIN {X 0,Y 261.078,Z 797.873,A -85,B 0,C 180,E1 -18470.69,E2 -18470.69} C_VEL
LIN {X 0,Y 262.781,Z 786.48,A -85,B 0,C 180,E1 -18472.195,E2 -18472.195} C_VEL
LIN {X 0,Y 264.309,Z 774.729,A -85,B 0,C 180,E1 -18473.402,E2 -18473.402} C_VEL
LIN {X 0,Y 265.675,Z 761.988,A -85,B 0,C 180,E1 -18474.362,E2 -18474.362} C_VEL
LIN {X 0,Y 266.689,Z 747.906,A -85,B 0,C 180,E1 -18475.086,E2 -18475.086} C_VEL
LIN {X 0,Y 268.659,Z 688.619,A -85,B 0,C 180,E1 -18476.879,E2 -18476.879} C_VEL
LIN {X 0,Y 263.103,Z 646.88,A -85,B 0,C 180,E1 -18478.749,E2 -18478.749} C_VEL
LIN {X 0,Y 260.508,Z 639.314,A -85,B 0,C 180,E1 -18479.259,E2 -18479.259} C_VEL
LIN {X 0,Y 258.075,Z 627.372,A -85,B 0,C 180,E1 -18483.466,E2 -18483.466} C_VEL
LIN {X 0,Y 256.174,Z 618.575,A -85,B 0,C 180,E1 -18486.755,E2 -18486.755} C_VEL
LIN {X 0,Y 256.084,Z 618.587,A -85,B 0,C 180,E1 -18491.196,E2 -18491.196} C_VEL
LIN {X 0,Y 256.071,Z 618.587,A -85,B 0,C 180,E1 -18495.526,E2 -18495.526} C_VEL
LIN {X 0,Y 256.083,Z 618.587,A -85,B 0,C 180,E1 -18498.801,E2 -18498.801} C_VEL
LIN {X 0,Y 256.152,Z 618.58,A -85,B 0,C 180,E1 -18502.87,E2 -18502.87} C_VEL
LIN {X 0,Y 256.083,Z 618.588,A -85,B 0,C 180,E1 -18506.709,E2 -18506.709} C_VEL
LIN {X 0,Y 256.135,Z 618.579,A -85,B 0,C 180,E1 -18511.404,E2 -18511.404} C_VEL
LIN {X 0,Y 256.139,Z 618.577,A -85,B 0,C 180,E1 -18515.695,E2 -18515.695} C_VEL
LIN {X 0,Y 256.158,Z 618.578,A -85,B 0,C 180,E1 -18519.103,E2 -18519.103} C_VEL
LIN {X 0,Y 256.29,Z 618.558,A -85,B 0,C 180,E1 -18524.084,E2 -18524.084} C_VEL
LIN {X 0,Y 256.304,Z 618.557,A -85,B 0,C 180,E1 -18528.933,E2 -18528.933} C_VEL
LIN {X 0,Y 256.532,Z 618.525,A -85,B 0,C 180,E1 -18532.126,E2 -18532.126} C_VEL
LIN {X 0,Y 256.709,Z 618.503,A -85,B 0,C 180,E1 -18538.43,E2 -18538.43} C_VEL
LIN {X 0,Y 256.709,Z 618.502,A -85,B 0,C 180,E1 -18541.568,E2 -18541.568} C_VEL
LIN {X 0,Y 256.532,Z 618.529,A -85,B 0,C 180,E1 -18547.872,E2 -18547.872} C_VEL
LIN {X 0,Y 256.303,Z 618.553,A -85,B 0,C 180,E1 -18551.065,E2 -18551.065} C_VEL
LIN {X 0,Y 256.273,Z 618.561,A -85,B 0,C 180,E1 -18555.916,E2 -18555.916} C_VEL
LIN {X 0,Y 256.16,Z 618.572,A -85,B 0,C 180,E1 -18560.895,E2 -18560.895} C_VEL
LIN {X 0,Y 256.182,Z 618.563,A -85,B 0,C 180,E1 -18565.138,E2 -18565.138} C_VEL
LIN {X 0,Y 256.098,Z 618.581,A -85,B 0,C 180,E1 -18569.601,E2 -18569.601} C_VEL
LIN {X 0,Y 256.079,Z 618.583,A -85,B 0,C 180,E1 -18573.29,E2 -18573.29} C_VEL
LIN {X 0,Y 256.135,Z 618.57,A -85,B 0,C 180,E1 -18577.278,E2 -18577.278} C_VEL
LIN {X 0,Y 256.098,Z 618.58,A -85,B 0,C 180,E1 -18581.194,E2 -18581.194} C_VEL
LIN {X 0,Y 256.071,Z 618.585,A -85,B 0,C 180,E1 -18585.526,E2 -18585.526} C_VEL
LIN {X 0,Y 256.081,Z 618.578,A -85,B 0,C 180,E1 -18588.803,E2 -18588.803} C_VEL
LIN {X 0,Y 256.149,Z 618.577,A -85,B 0,C 180,E1 -18592.872,E2 -18592.872} C_VEL
LIN {X 0,Y 256.08,Z 618.585,A -85,B 0,C 180,E1 -18596.71,E2 -18596.71} C_VEL
LIN {X 0,Y 256.122,Z 618.578,A -85,B 0,C 180,E1 -18601.41,E2 -18601.41} C_VEL
LIN {X 0,Y 256.163,Z 618.573,A -85,B 0,C 180,E1 -18605.699,E2 -18605.699} C_VEL
LIN {X 0,Y 256.163,Z 618.575,A -85,B 0,C 180,E1 -18609.105,E2 -18609.105} C_VEL
LIN {X 0,Y 256.296,Z 618.557,A -85,B 0,C 180,E1 -18614.085,E2 -18614.085} C_VEL
LIN {X 0,Y 256.307,Z 618.558,A -85,B 0,C 180,E1 -18618.934,E2 -18618.934} C_VEL
LIN {X 0,Y 256.534,Z 618.525,A -85,B 0,C 180,E1 -18622.127,E2 -18622.127} C_VEL
LIN {X 0,Y 256.712,Z 618.505,A -85,B 0,C 180,E1 -18628.431,E2 -18628.431} C_VEL
LIN {X 0,Y 256.712,Z 618.506,A -85,B 0,C 180,E1 -18631.569,E2 -18631.569} C_VEL
LIN {X 0,Y 256.479,Z 618.535,A -85,B 0,C 180,E1 -18636.293,E2 -18636.293} C_VEL
LIN {X 0,Y 256.423,Z 618.545,A -85,B 0,C 180,E1 -18639.465,E2 -18639.465} C_VEL
LIN {X 0,Y 256.252,Z 618.566,A -85,B 0,C 180,E1 -18644.29,E2 -18644.29} C_VEL
LIN {X 0,Y 256.314,Z 618.56,A -85,B 0,C 180,E1 -18645.506,E2 -18645.506} C_VEL
LIN {X 0,Y 257.5,Z 621.804,A -85,B 0,C 180,E1 -18645.762,E2 -18645.762} C_VEL
LIN {X 0,Y 263.418,Z 635.783,A -85,B 0,C 180,E1 -18646.803,E2 -18646.803} C_VEL
LIN {X 0,Y 269.624,Z 652.928,A -85,B 0,C 180,E1 -18647.926,E2 -18647.926} C_VEL
LIN {X 0,Y 266.978,Z 722.927,A -85,B 0,C 180,E1 -18650.011,E2 -18650.011} C_VEL
LIN {X 0,Y 266.145,Z 736.781,A -85,B 0,C 180,E1 -18650.733,E2 -18650.733} C_VEL
LIN {X 0,Y 265.06,Z 749.315,A -85,B 0,C 180,E1 -18651.683,E2 -18651.683} C_VEL
LIN {X 0,Y 263.701,Z 761.512,A -85,B 0,C 180,E1 -18652.94,E2 -18652.94} C_VEL
LIN {X 0,Y 262.28,Z 772.231,A -85,B 0,C 180,E1 -18654.35,E2 -18654.35} C_VEL
LIN {X 0,Y 260.727,Z 782.214,A -85,B 0,C 180,E1 -18655.977,E2 -18655.977} C_VEL
LIN {X 0,Y 259.263,Z 791.601,A -85,B 0,C 180,E1 -18657.878,E2 -18657.878} C_VEL
LIN {X 0,Y 257.953,Z 799.404,A -85,B 0,C 180,E1 -18659.815,E2 -18659.815} C_VEL
LIN {X 0,Y 256.768,Z 806.451,A -85,B 0,C 180,E1 -18661.953,E2 -18661.953} C_VEL
LIN {X 0,Y 255.688,Z 813.045,A -85,B 0,C 180,E1 -18664.454,E2 -18664.454} C_VEL
LIN {X 0,Y 254.966,Z 818.129,A -85,B 0,C 180,E1 -18666.932,E2 -18666.932} C_VEL
LIN {X 0,Y 254.337,Z 822.034,A -85,B 0,C 180,E1 -18669.46,E2 -18669.46} C_VEL
LIN {X 0,Y 254.008,Z 824.454,A -85,B 0,C 180,E1 -18671.666,E2 -18671.666} C_VEL
LIN {X 0,Y 253.863,Z 826.101,A -85,B 0,C 180,E1 -18673.964,E2 -18673.964} C_VEL
LIN {X 0,Y 253.889,Z 826.884,A -85,B 0,C 180,E1 -18676.21,E2 -18676.21} C_VEL
LIN {X 0,Y 254.107,Z 826.883,A -85,B 0,C 180,E1 -18678.412,E2 -18678.412} C_VEL
LIN {X 0,Y 254.574,Z 826.078,A -85,B 0,C 180,E1 -18680.622,E2 -18680.622} C_VEL
LIN {X 0,Y 255.258,Z 824.33,A -85,B 0,C 180,E1 -18682.981,E2 -18682.981} C_VEL
LIN {X 0,Y 256.174,Z 821.574,A -85,B 0,C 180,E1 -18685.388,E2 -18685.388} C_VEL
LIN {X 0,Y 257.44,Z 817.702,A -85,B 0,C 180,E1 -18687.808,E2 -18687.808} C_VEL
LIN {X 0,Y 259.052,Z 812.557,A -85,B 0,C 180,E1 -18690.242,E2 -18690.242} C_VEL
LIN {X 0,Y 261.189,Z 805.546,A -85,B 0,C 180,E1 -18692.78,E2 -18692.78} C_VEL
LIN {X 0,Y 263.542,Z 797.552,A -85,B 0,C 180,E1 -18695.049,E2 -18695.049} C_VEL
LIN {X 0,Y 265.965,Z 788.53,A -85,B 0,C 180,E1 -18697.092,E2 -18697.092} C_VEL
LIN {X 0,Y 268.514,Z 777.79,A -85,B 0,C 180,E1 -18699.004,E2 -18699.004} C_VEL
LIN {X 0,Y 270.76,Z 767.305,A -85,B 0,C 180,E1 -18700.478,E2 -18700.478} C_VEL
LIN {X 0,Y 272.855,Z 755.263,A -85,B 0,C 180,E1 -18701.803,E2 -18701.803} C_VEL
LIN {X 0,Y 274.643,Z 742.062,A -85,B 0,C 180,E1 -18702.886,E2 -18702.886} C_VEL
LIN {X 0,Y 275.744,Z 730.462,A -85,B 0,C 180,E1 -18703.576,E2 -18703.576} C_VEL
LIN {X 0,Y 276.656,Z 717.082,A -85,B 0,C 180,E1 -18704.073,E2 -18704.073} C_VEL
LIN {X 0,Y 279.552,Z 661.651,A -85,B 0,C 180,E1 -18705.735,E2 -18705.735} C_VEL
LIN {X 0,Y 274.469,Z 650.234,A -85,B 0,C 180,E1 -18707.054,E2 -18707.054} C_VEL
LIN {X 0,Y 269.122,Z 640.099,A -85,B 0,C 180,E1 -18708.489,E2 -18708.489} C_VEL
LIN {X 0,Y 264.242,Z 631.969,A -85,B 0,C 180,E1 -18709.849,E2 -18709.849} C_VEL
LIN {X 0,Y 260.469,Z 625.843,A -85,B 0,C 180,E1 -18710.974,E2 -18710.974} C_VEL
LIN {X 0,Y 258.997,Z 623.701,A -85,B 0,C 180,E1 -18711.424,E2 -18711.424} C_VEL
LIN {X 0,Y 256.193,Z 622.029,A -85,B 0,C 180,E1 -18712.185,E2 -18712.185} C_VEL
LIN {X 0,Y 250.486,Z 620.723,A -85,B 0,C 180,E1 -18713.953,E2 -18713.953} C_VEL
LIN {X 0,Y 249.462,Z 620.015,A -85,B 0,C 180,E1 -18714.685,E2 -18714.685} C_VEL
LIN {X 0,Y 249.398,Z 619.817,A -85,B 0,C 180,E1 -18714.835,E2 -18714.835} C_VEL
LIN {X 0,Y 249.31,Z 619.431,A -85,B 0,C 180,E1 -18715.15,E2 -18715.15} C_VEL
LIN {X 0,Y 249.679,Z 619.381,A -85,B 0,C 180,E1 -18718.388,E2 -18718.388} C_VEL
LIN {X 0,Y 249.673,Z 619.381,A -85,B 0,C 180,E1 -18721.614,E2 -18721.614} C_VEL
LIN {X 0,Y 249.457,Z 619.406,A -85,B 0,C 180,E1 -18726.471,E2 -18726.471} C_VEL
LIN {X 0,Y 249.384,Z 619.414,A -85,B 0,C 180,E1 -18729.736,E2 -18729.736} C_VEL
LIN {X 0,Y 249.197,Z 619.444,A -85,B 0,C 180,E1 -18734.705,E2 -18734.705} C_VEL
LIN {X 0,Y 249.135,Z 619.451,A -85,B 0,C 180,E1 -18738.079,E2 -18738.079} C_VEL
LIN {X 0,Y 249.084,Z 619.455,A -85,B 0,C 180,E1 -18741.519,E2 -18741.519} C_VEL
LIN {X 0,Y 249.127,Z 619.443,A -85,B 0,C 180,E1 -18745.483,E2 -18745.483} C_VEL
LIN {X 0,Y 249.071,Z 619.449,A -85,B 0,C 180,E1 -18748.99,E2 -18748.99} C_VEL
LIN {X 0,Y 249.034,Z 619.453,A -85,B 0,C 180,E1 -18752.426,E2 -18752.426} C_VEL
LIN {X 0,Y 249.072,Z 619.457,A -85,B 0,C 180,E1 -18756.339,E2 -18756.339} C_VEL
LIN {X 0,Y 249.036,Z 619.458,A -85,B 0,C 180,E1 -18760.473,E2 -18760.473} C_VEL
LIN {X 0,Y 249.089,Z 619.646,A -85,B 0,C 180,E1 -18762.934,E2 -18762.934} C_VEL
LIN {X 0,Y 250.867,Z 625.42,A -85,B 0,C 180,E1 -18766.752,E2 -18766.752} C_VEL
LIN {X 0,Y 252.655,Z 631.432,A -85,B 0,C 180,E1 -18770.226,E2 -18770.226} C_VEL
LIN {X 0,Y 253.596,Z 635.123,A -85,B 0,C 180,E1 -18772.099,E2 -18772.099} C_VEL
LIN {X 0,Y 256.118,Z 639.698,A -85,B 0,C 180,E1 -18772.945,E2 -18772.945} C_VEL
LIN {X 0,Y 260.333,Z 647.389,A -85,B 0,C 180,E1 -18774.285,E2 -18774.285} C_VEL
LIN {X 0,Y 264.445,Z 655.492,A -85,B 0,C 180,E1 -18775.524,E2 -18775.524} C_VEL
LIN {X 0,Y 269.351,Z 666.545,A -85,B 0,C 180,E1 -18776.957,E2 -18776.957} C_VEL
LIN {X 0,Y 271.772,Z 683.313,A -85,B 0,C 180,E1 -18778.08,E2 -18778.08} C_VEL
LIN {X 0,Y 272.655,Z 692.824,A -85,B 0,C 180,E1 -18778.61,E2 -18778.61} C_VEL
LIN {X 0,Y 269.712,Z 746.011,A -85,B 0,C 180,E1 -18780.268,E2 -18780.268} C_VEL
LIN {X 0,Y 268.126,Z 760.332,A -85,B 0,C 180,E1 -18780.994,E2 -18780.994} C_VEL
LIN {X 0,Y 266.26,Z 772.065,A -85,B 0,C 180,E1 -18781.849,E2 -18781.849} C_VEL
LIN {X 0,Y 263.895,Z 784.415,A -85,B 0,C 180,E1 -18783.081,E2 -18783.081} C_VEL
LIN {X 0,Y 261.397,Z 795.622,A -85,B 0,C 180,E1 -18784.522,E2 -18784.522} C_VEL
LIN {X 0,Y 258.77,Z 805.841,A -85,B 0,C 180,E1 -18786.173,E2 -18786.173} C_VEL
LIN {X 0,Y 255.981,Z 815.914,A -85,B 0,C 180,E1 -18788.245,E2 -18788.245} C_VEL
LIN {X 0,Y 253.484,Z 824.844,A -85,B 0,C 180,E1 -18790.567,E2 -18790.567} C_VEL
LIN {X 0,Y 251.443,Z 832.05,A -85,B 0,C 180,E1 -18792.934,E2 -18792.934} C_VEL
LIN {X 0,Y 249.686,Z 837.855,A -85,B 0,C 180,E1 -18795.326,E2 -18795.326} C_VEL
LIN {X 0,Y 248.378,Z 842.483,A -85,B 0,C 180,E1 -18797.748,E2 -18797.748} C_VEL
LIN {X 0,Y 247.588,Z 846.034,A -85,B 0,C 180,E1 -18800.194,E2 -18800.194} C_VEL
LIN {X 0,Y 247.063,Z 849.214,A -85,B 0,C 180,E1 -18803.467,E2 -18803.467} C_VEL
LIN {X 0,Y 246.973,Z 850.203,A -85,B 0,C 180,E1 -18805.103,E2 -18805.103} C_VEL
LIN {X 0,Y 247.007,Z 850.751,A -85,B 0,C 180,E1 -18806.738,E2 -18806.738} C_VEL
LIN {X 0,Y 247.058,Z 850.886,A -85,B 0,C 180,E1 -18808.37,E2 -18808.37} C_VEL
LIN {X 0,Y 247.115,Z 850.62,A -85,B 0,C 180,E1 -18810,E2 -18810} C_VEL
LIN {X 0,Y 247.08,Z 849.943,A -85,B 0,C 180,E1 -18811.63,E2 -18811.63} C_VEL
LIN {X 0,Y 247.059,Z 848.801,A -85,B 0,C 180,E1 -18813.261,E2 -18813.261} C_VEL
LIN {X 0,Y 247.031,Z 846.788,A -85,B 0,C 180,E1 -18815.28,E2 -18815.28} C_VEL
LIN {X 0,Y 247.276,Z 842.664,A -85,B 0,C 180,E1 -18818.17,E2 -18818.17} C_VEL
LIN {X 0,Y 247.749,Z 837.891,A -85,B 0,C 180,E1 -18820.625,E2 -18820.625} C_VEL
LIN {X 0,Y 248.749,Z 830.669,A -85,B 0,C 180,E1 -18823.479,E2 -18823.479} C_VEL
LIN {X 0,Y 249.797,Z 824.211,A -85,B 0,C 180,E1 -18825.502,E2 -18825.502} C_VEL
LIN {X 0,Y 250.858,Z 818.132,A -85,B 0,C 180,E1 -18827.1,E2 -18827.1} C_VEL
LIN {X 0,Y 251.767,Z 812.275,A -85,B 0,C 180,E1 -18828.439,E2 -18828.439} C_VEL
LIN {X 0,Y 253.333,Z 802.565,A -85,B 0,C 180,E1 -18830.29,E2 -18830.29} C_VEL
LIN {X 0,Y 254.967,Z 792.382,A -85,B 0,C 180,E1 -18831.846,E2 -18831.846} C_VEL
LIN {X 0,Y 256.636,Z 781.357,A -85,B 0,C 180,E1 -18833.182,E2 -18833.182} C_VEL
LIN {X 0,Y 258.155,Z 769.244,A -85,B 0,C 180,E1 -18834.315,E2 -18834.315} C_VEL
LIN {X 0,Y 259.461,Z 755.927,A -85,B 0,C 180,E1 -18835.199,E2 -18835.199} C_VEL
LIN {X 0,Y 260.239,Z 742.527,A -85,B 0,C 180,E1 -18835.779,E2 -18835.779} C_VEL
LIN {X 0,Y 262.017,Z 689.358,A -85,B 0,C 180,E1 -18837.408,E2 -18837.408} C_VEL
LIN {X 0,Y 256.712,Z 648.948,A -85,B 0,C 180,E1 -18839.272,E2 -18839.272} C_VEL
LIN {X 0,Y 253.216,Z 638.978,A -85,B 0,C 180,E1 -18839.972,E2 -18839.972} C_VEL
LIN {X 0,Y 250.534,Z 625.902,A -85,B 0,C 180,E1 -18844.746,E2 -18844.746} C_VEL
LIN {X 0,Y 249.093,Z 619.455,A -85,B 0,C 180,E1 -18847.28,E2 -18847.28} C_VEL
LIN {X 0,Y 249.044,Z 619.466,A -85,B 0,C 180,E1 -18850.469,E2 -18850.469} C_VEL
LIN {X 0,Y 249.044,Z 619.466,A -85,B 0,C 180,E1 -18852.8,E2 -18852.8} C_VEL
LIN {X 0,Y 249.038,Z 619.463,A -85,B 0,C 180,E1 -18857.367,E2 -18857.367} C_VEL
LIN {X 0,Y 249.05,Z 619.46,A -85,B 0,C 180,E1 -18861.623,E2 -18861.623} C_VEL
LIN {X 0,Y 249.059,Z 619.46,A -85,B 0,C 180,E1 -18865.641,E2 -18865.641} C_VEL
LIN {X 0,Y 249.05,Z 619.46,A -85,B 0,C 180,E1 -18869.472,E2 -18869.472} C_VEL
LIN {X 0,Y 249.067,Z 619.458,A -85,B 0,C 180,E1 -18873.161,E2 -18873.161} C_VEL
LIN {X 0,Y 249.057,Z 619.461,A -85,B 0,C 180,E1 -18876.73,E2 -18876.73} C_VEL
LIN {X 0,Y 249.103,Z 619.452,A -85,B 0,C 180,E1 -18880.21,E2 -18880.21} C_VEL
LIN {X 0,Y 249.238,Z 619.438,A -85,B 0,C 180,E1 -18883.621,E2 -18883.621} C_VEL
LIN {X 0,Y 249.247,Z 619.435,A -85,B 0,C 180,E1 -18888.616,E2 -18888.616} C_VEL
LIN {X 0,Y 249.474,Z 619.405,A -85,B 0,C 180,E1 -18891.902,E2 -18891.902} C_VEL
LIN {X 0,Y 249.431,Z 619.413,A -85,B 0,C 180,E1 -18896.769,E2 -18896.769} C_VEL
LIN {X 0,Y 249.729,Z 619.369,A -85,B 0,C 180,E1 -18899.999,E2 -18899.999} C_VEL
LIN {X 0,Y 249.431,Z 619.409,A -85,B 0,C 180,E1 -18903.23,E2 -18903.23} C_VEL
LIN {X 0,Y 249.474,Z 619.407,A -85,B 0,C 180,E1 -18908.097,E2 -18908.097} C_VEL
LIN {X 0,Y 249.246,Z 619.434,A -85,B 0,C 180,E1 -18911.383,E2 -18911.383} C_VEL
LIN {X 0,Y 249.212,Z 619.437,A -85,B 0,C 180,E1 -18916.503,E2 -18916.503} C_VEL
LIN {X 0,Y 249.081,Z 619.456,A -85,B 0,C 180,E1 -18921.518,E2 -18921.518} C_VEL
LIN {X 0,Y 249.124,Z 619.442,A -85,B 0,C 180,E1 -18925.482,E2 -18925.482} C_VEL
LIN {X 0,Y 249.067,Z 619.454,A -85,B 0,C 180,E1 -18928.989,E2 -18928.989} C_VEL
LIN {X 0,Y 249.03,Z 619.463,A -85,B 0,C 180,E1 -18932.425,E2 -18932.425} C_VEL
LIN {X 0,Y 249.069,Z 619.452,A -85,B 0,C 180,E1 -18936.338,E2 -18936.338} C_VEL
LIN {X 0,Y 249.072,Z 619.457,A -85,B 0,C 180,E1 -18940.464,E2 -18940.464} C_VEL
LIN {X 0,Y 249.017,Z 619.464,A -85,B 0,C 180,E1 -18944.875,E2 -18944.875} C_VEL
LIN {X 0,Y 249.049,Z 619.457,A -85,B 0,C 180,E1 -18947.371,E2 -18947.371} C_VEL
LIN {X 0,Y 249.06,Z 619.458,A -85,B 0,C 180,E1 -18952.194,E2 -18952.194} C_VEL
LIN {X 0,Y 249.057,Z 619.459,A -85,B 0,C 180,E1 -18955.642,E2 -18955.642} C_VEL
LIN {X 0,Y 249.043,Z 619.454,A -85,B 0,C 180,E1 -18959.473,E2 -18959.473} C_VEL
LIN {X 0,Y 249.067,Z 619.459,A -85,B 0,C 180,E1 -18963.162,E2 -18963.162} C_VEL
LIN {X 0,Y 249.076,Z 619.461,A -85,B 0,C 180,E1 -18966.733,E2 -18966.733} C_VEL
LIN {X 0,Y 249.107,Z 619.453,A -85,B 0,C 180,E1 -18970.212,E2 -18970.212} C_VEL
LIN {X 0,Y 249.239,Z 619.436,A -85,B 0,C 180,E1 -18973.622,E2 -18973.622} C_VEL
LIN {X 0,Y 249.25,Z 619.436,A -85,B 0,C 180,E1 -18978.617,E2 -18978.617} C_VEL
LIN {X 0,Y 249.477,Z 619.404,A -85,B 0,C 180,E1 -18981.903,E2 -18981.903} C_VEL
LIN {X 0,Y 249.434,Z 619.413,A -85,B 0,C 180,E1 -18986.77,E2 -18986.77} C_VEL
LIN {X 0,Y 249.726,Z 619.374,A -85,B 0,C 180,E1 -18990,E2 -18990} C_VEL
LIN {X 0,Y 249.434,Z 619.415,A -85,B 0,C 180,E1 -18993.23,E2 -18993.23} C_VEL
LIN {X 0,Y 249.451,Z 619.41,A -85,B 0,C 180,E1 -18996.471,E2 -18996.471} C_VEL
LIN {X 0,Y 249.34,Z 619.426,A -85,B 0,C 180,E1 -18999.736,E2 -18999.736} C_VEL
LIN {X 0,Y 249.259,Z 619.589,A -85,B 0,C 180,E1 -19004.856,E2 -19004.856} C_VEL
LIN {X 0,Y 250.363,Z 622.48,A -85,B 0,C 180,E1 -19005.075,E2 -19005.075} C_VEL
LIN {X 0,Y 257.139,Z 638.085,A -85,B 0,C 180,E1 -19006.297,E2 -19006.297} C_VEL
LIN {X 0,Y 263.058,Z 654.596,A -85,B 0,C 180,E1 -19007.404,E2 -19007.404} C_VEL
LIN {X 0,Y 260.274,Z 724.239,A -85,B 0,C 180,E1 -19009.542,E2 -19009.542} C_VEL
